LIN {X 0,Y 304.577,Z 613.756,A -85,B 0,C 180,E1 -15941.986,E2 -15941.986} C_VEL
LIN {X 0,Y 305.536,Z 607.014,A -85,B 0,C 180,E1 -15944.657,E2 -15944.657} C_VEL
LIN {X 0,Y 306.864,Z 599.737,A -85,B 0,C 180,E1 -15946.978,E2 -15946.978} C_VEL
LIN {X 0,Y 308.524,Z 590.973,A -85,B 0,C 180,E1 -15949.287,E2 -15949.287} C_VEL
LIN {X 0,Y 310.431,Z 582.076,A -85,B 0,C 180,E1 -15951.237,E2 -15951.237} C_VEL
LIN {X 0,Y 312.411,Z 571.551,A -85,B 0,C 180,E1 -15953.184,E2 -15953.184} C_VEL
LIN {X 0,Y 314.648,Z 560.119,A -85,B 0,C 180,E1 -15954.935,E2 -15954.935} C_VEL
LIN {X 0,Y 316.992,Z 547.692,A -85,B 0,C 180,E1 -15956.499,E2 -15956.499} C_VEL
LIN {X 0,Y 319.156,Z 534.543,A -85,B 0,C 180,E1 -15957.854,E2 -15957.854} C_VEL
LIN {X 0,Y 321.209,Z 520.123,A -85,B 0,C 180,E1 -15959.042,E2 -15959.042} C_VEL
LIN {X 0,Y 322.937,Z 505.843,A -85,B 0,C 180,E1 -15959.946,E2 -15959.946} C_VEL
LIN {X 0,Y 324.415,Z 490.603,A -85,B 0,C 180,E1 -15960.648,E2 -15960.648} C_VEL
LIN {X 0,Y 325.39,Z 474.711,A -85,B 0,C 180,E1 -15961.132,E2 -15961.132} C_VEL
LIN {X 0,Y 329.171,Z 367.113,A -85,B 0,C 180,E1 -15963.574,E2 -15963.574} C_VEL
LIN {X 0,Y 326.556,Z 352.02,A -85,B 0,C 180,E1 -15964.25,E2 -15964.25} C_VEL
LIN {X 0,Y 317.025,Z 330.376,A -85,B 0,C 180,E1 -15965.899,E2 -15965.899} C_VEL
LIN {X 0,Y 309.608,Z 314.884,A -85,B 0,C 180,E1 -15967.238,E2 -15967.238} C_VEL
LIN {X 0,Y 306.205,Z 302.97,A -85,B 0,C 180,E1 -15970.761,E2 -15970.761} C_VEL
LIN {X 0,Y 305.417,Z 300.068,A -85,B 0,C 180,E1 -15971.691,E2 -15971.691} C_VEL
LIN {X 0,Y 305.401,Z 300.067,A -85,B 0,C 180,E1 -15975.51,E2 -15975.51} C_VEL
LIN {X 0,Y 305.413,Z 300.072,A -85,B 0,C 180,E1 -15978.137,E2 -15978.137} C_VEL
LIN {X 0,Y 305.443,Z 300.059,A -85,B 0,C 180,E1 -15981.591,E2 -15981.591} C_VEL
LIN {X 0,Y 305.462,Z 300.049,A -85,B 0,C 180,E1 -15984.885,E2 -15984.885} C_VEL
LIN {X 0,Y 305.443,Z 300.063,A -85,B 0,C 180,E1 -15988.357,E2 -15988.357} C_VEL
LIN {X 0,Y 305.461,Z 300.061,A -85,B 0,C 180,E1 -15991.106,E2 -15991.106} C_VEL
LIN {X 0,Y 305.479,Z 300.062,A -85,B 0,C 180,E1 -15994.078,E2 -15994.078} C_VEL
LIN {X 0,Y 305.462,Z 300.065,A -85,B 0,C 180,E1 -15998.398,E2 -15998.398} C_VEL
LIN {X 0,Y 305.534,Z 300.055,A -85,B 0,C 180,E1 -16002.599,E2 -16002.599} C_VEL
LIN {X 0,Y 305.624,Z 300.022,A -85,B 0,C 180,E1 -16005.346,E2 -16005.346} C_VEL
LIN {X 0,Y 305.619,Z 300.022,A -85,B 0,C 180,E1 -16009.397,E2 -16009.397} C_VEL
LIN {X 0,Y 305.735,Z 300.026,A -85,B 0,C 180,E1 -16012.07,E2 -16012.07} C_VEL
LIN {X 0,Y 305.648,Z 300.023,A -85,B 0,C 180,E1 -16014.721,E2 -16014.721} C_VEL
LIN {X 0,Y 305.935,Z 299.985,A -85,B 0,C 180,E1 -16018.682,E2 -16018.682} C_VEL
LIN {X 0,Y 305.929,Z 300.002,A -85,B 0,C 180,E1 -16021.314,E2 -16021.314} C_VEL
LIN {X 0,Y 305.642,Z 300.007,A -85,B 0,C 180,E1 -16025.275,E2 -16025.275} C_VEL
LIN {X 0,Y 305.726,Z 299.997,A -85,B 0,C 180,E1 -16027.926,E2 -16027.926} C_VEL
LIN {X 0,Y 305.588,Z 300.044,A -85,B 0,C 180,E1 -16031.943,E2 -16031.943} C_VEL
LIN {X 0,Y 305.601,Z 300.02,A -85,B 0,C 180,E1 -16035.011,E2 -16035.011} C_VEL
LIN {X 0,Y 305.534,Z 300.035,A -85,B 0,C 180,E1 -16039.424,E2 -16039.424} C_VEL
LIN {X 0,Y 305.447,Z 300.062,A -85,B 0,C 180,E1 -16043.023,E2 -16043.023} C_VEL
LIN {X 0,Y 305.44,Z 300.031,A -85,B 0,C 180,E1 -16046.187,E2 -16046.187} C_VEL
LIN {X 0,Y 305.413,Z 300.045,A -85,B 0,C 180,E1 -16049.023,E2 -16049.023} C_VEL
LIN {X 0,Y 305.425,Z 300.064,A -85,B 0,C 180,E1 -16051.951,E2 -16051.951} C_VEL
LIN {X 0,Y 305.449,Z 300.04,A -85,B 0,C 180,E1 -16055.112,E2 -16055.112} C_VEL
LIN {X 0,Y 305.421,Z 300.049,A -85,B 0,C 180,E1 -16058.523,E2 -16058.523} C_VEL
LIN {X 0,Y 305.422,Z 300.064,A -85,B 0,C 180,E1 -16062.58,E2 -16062.58} C_VEL
LIN {X 0,Y 305.411,Z 300.047,A -85,B 0,C 180,E1 -16066.343,E2 -16066.343} C_VEL
LIN {X 0,Y 305.444,Z 300.063,A -85,B 0,C 180,E1 -16069.891,E2 -16069.891} C_VEL
LIN {X 0,Y 305.45,Z 300.044,A -85,B 0,C 180,E1 -16073.634,E2 -16073.634} C_VEL
LIN {X 0,Y 305.45,Z 300.064,A -85,B 0,C 180,E1 -16076.482,E2 -16076.482} C_VEL
LIN {X 0,Y 305.465,Z 300.05,A -85,B 0,C 180,E1 -16080.954,E2 -16080.954} C_VEL
LIN {X 0,Y 305.555,Z 300.041,A -85,B 0,C 180,E1 -16084.087,E2 -16084.087} C_VEL
LIN {X 0,Y 305.466,Z 300.058,A -85,B 0,C 180,E1 -16088.4,E2 -16088.4} C_VEL
LIN {X 0,Y 305.564,Z 300.051,A -85,B 0,C 180,E1 -16091.216,E2 -16091.216} C_VEL
LIN {X 0,Y 305.633,Z 300.039,A -85,B 0,C 180,E1 -16095.348,E2 -16095.348} C_VEL
LIN {X 0,Y 305.624,Z 300.035,A -85,B 0,C 180,E1 -16099.399,E2 -16099.399} C_VEL
LIN {X 0,Y 305.807,Z 300.029,A -85,B 0,C 180,E1 -16102.323,E2 -16102.323} C_VEL
LIN {X 0,Y 306.955,Z 303.051,A -85,B 0,C 180,E1 -16102.591,E2 -16102.591} C_VEL
LIN {X 0,Y 308.436,Z 305.417,A -85,B 0,C 180,E1 -16102.849,E2 -16102.849} C_VEL
LIN {X 0,Y 312.255,Z 312.818,A -85,B 0,C 180,E1 -16103.538,E2 -16103.538} C_VEL
LIN {X 0,Y 320.275,Z 328.458,A -85,B 0,C 180,E1 -16104.919,E2 -16104.919} C_VEL
LIN {X 0,Y 327.005,Z 343.478,A -85,B 0,C 180,E1 -16106.065,E2 -16106.065} C_VEL
LIN {X 0,Y 329.522,Z 349.607,A -85,B 0,C 180,E1 -16106.495,E2 -16106.495} C_VEL
LIN {X 0,Y 325.777,Z 455.006,A -85,B 0,C 180,E1 -16108.879,E2 -16108.879} C_VEL
LIN {X 0,Y 324.99,Z 471.109,A -85,B 0,C 180,E1 -16109.341,E2 -16109.341} C_VEL
LIN {X 0,Y 323.73,Z 486.619,A -85,B 0,C 180,E1 -16110.029,E2 -16110.029} C_VEL
LIN {X 0,Y 322.104,Z 501.197,A -85,B 0,C 180,E1 -16110.922,E2 -16110.922} C_VEL
LIN {X 0,Y 320.359,Z 515.115,A -85,B 0,C 180,E1 -16112.042,E2 -16112.042} C_VEL
LIN {X 0,Y 318.327,Z 527.994,A -85,B 0,C 180,E1 -16113.322,E2 -16113.322} C_VEL
LIN {X 0,Y 316.161,Z 540.387,A -85,B 0,C 180,E1 -16114.828,E2 -16114.828} C_VEL
LIN {X 0,Y 313.949,Z 552.293,A -85,B 0,C 180,E1 -16116.587,E2 -16116.587} C_VEL
LIN {X 0,Y 311.841,Z 562.917,A -85,B 0,C 180,E1 -16118.476,E2 -16118.476} C_VEL
LIN {X 0,Y 309.656,Z 573.654,A -85,B 0,C 180,E1 -16120.791,E2 -16120.791} C_VEL
LIN {X 0,Y 307.746,Z 582.782,A -85,B 0,C 180,E1 -16123.2,E2 -16123.2} C_VEL
LIN {X 0,Y 306.329,Z 589.979,A -85,B 0,C 180,E1 -16125.521,E2 -16125.521} C_VEL
LIN {X 0,Y 305.184,Z 596.469,A -85,B 0,C 180,E1 -16128.112,E2 -16128.112} C_VEL
LIN {X 0,Y 304.506,Z 600.773,A -85,B 0,C 180,E1 -16130.254,E2 -16130.254} C_VEL
LIN {X 0,Y 304.024,Z 604.144,A -85,B 0,C 180,E1 -16132.391,E2 -16132.391} C_VEL
LIN {X 0,Y 303.484,Z 607.573,A -85,B 0,C 180,E1 -16135.432,E2 -16135.432} C_VEL
LIN {X 0,Y 303.276,Z 609.377,A -85,B 0,C 180,E1 -16138.292,E2 -16138.292} C_VEL
LIN {X 0,Y 303.287,Z 609.865,A -85,B 0,C 180,E1 -16140.981,E2 -16140.981} C_VEL
LIN {X 0,Y 303.443,Z 609.138,A -85,B 0,C 180,E1 -16143.768,E2 -16143.768} C_VEL
LIN {X 0,Y 303.721,Z 607.678,A -85,B 0,C 180,E1 -16145.92,E2 -16145.92} C_VEL
LIN {X 0,Y 304.272,Z 604.832,A -85,B 0,C 180,E1 -16148.581,E2 -16148.581} C_VEL
LIN {X 0,Y 305.088,Z 600.978,A -85,B 0,C 180,E1 -16151.117,E2 -16151.117} C_VEL
LIN {X 0,Y 306.161,Z 596.204,A -85,B 0,C 180,E1 -16153.522,E2 -16153.522} C_VEL
LIN {X 0,Y 307.867,Z 588.815,A -85,B 0,C 180,E1 -16156.419,E2 -16156.419} C_VEL
LIN {X 0,Y 309.828,Z 580.921,A -85,B 0,C 180,E1 -16158.87,E2 -16158.87} C_VEL
LIN {X 0,Y 312.17,Z 571.322,A -85,B 0,C 180,E1 -16161.289,E2 -16161.289} C_VEL
LIN {X 0,Y 314.85,Z 560.656,A -85,B 0,C 180,E1 -16163.471,E2 -16163.471} C_VEL
LIN {X 0,Y 315.34,Z 558.594,A -85,B 0,C 180,E1 -16163.84,E2 -16163.84} C_VEL
LIN {X 0,Y 315.768,Z 554.512,A -85,B 0,C 180,E1 -16164.61,E2 -16164.61} C_VEL
LIN {X 0,Y 314.792,Z 547.859,A -85,B 0,C 180,E1 -16165.94,E2 -16165.94} C_VEL
LIN {X 0,Y 313.825,Z 540.87,A -85,B 0,C 180,E1 -16167.207,E2 -16167.207} C_VEL
LIN {X 0,Y 314.234,Z 536.226,A -85,B 0,C 180,E1 -16167.866,E2 -16167.866} C_VEL
LIN {X 0,Y 316.764,Z 523.451,A -85,B 0,C 180,E1 -16169.319,E2 -16169.319} C_VEL
LIN {X 0,Y 319.172,Z 509.538,A -85,B 0,C 180,E1 -16170.589,E2 -16170.589} C_VEL
LIN {X 0,Y 321.16,Z 495.876,A -85,B 0,C 180,E1 -16171.57,E2 -16171.57} C_VEL
LIN {X 0,Y 322.848,Z 481.049,A -85,B 0,C 180,E1 -16172.378,E2 -16172.378} C_VEL
LIN {X 0,Y 324.161,Z 465.241,A -85,B 0,C 180,E1 -16172.968,E2 -16172.968} C_VEL
LIN {X 0,Y 329.009,Z 355.514,A -85,B 0,C 180,E1 -16175.564,E2 -16175.564} C_VEL
LIN {X 0,Y 322.304,Z 340.991,A -85,B 0,C 180,E1 -16177.02,E2 -16177.02} C_VEL
LIN {X 0,Y 315.332,Z 328.219,A -85,B 0,C 180,E1 -16178.583,E2 -16178.583} C_VEL
LIN {X 0,Y 308.492,Z 316.768,A -85,B 0,C 180,E1 -16180.219,E2 -16180.219} C_VEL
LIN {X 0,Y 301.733,Z 306.632,A -85,B 0,C 180,E1 -16181.938,E2 -16181.938} C_VEL
LIN {X 0,Y 299.049,Z 302.887,A -85,B 0,C 180,E1 -16182.655,E2 -16182.655} C_VEL
LIN {X 0,Y 298.75,Z 302.016,A -85,B 0,C 180,E1 -16182.902,E2 -16182.902} C_VEL
LIN {X 0,Y 298.506,Z 300.928,A -85,B 0,C 180,E1 -16183.416,E2 -16183.416} C_VEL
LIN {X 0,Y 298.54,Z 300.924,A -85,B 0,C 180,E1 -16186.387,E2 -16186.387} C_VEL
LIN {X 0,Y 298.717,Z 300.898,A -85,B 0,C 180,E1 -16191.157,E2 -16191.157} C_VEL
LIN {X 0,Y 298.776,Z 300.891,A -85,B 0,C 180,E1 -16193.248,E2 -16193.248} C_VEL
LIN {X 0,Y 298.913,Z 300.873,A -85,B 0,C 180,E1 -16198.655,E2 -16198.655} C_VEL
LIN {X 0,Y 298.913,Z 300.872,A -85,B 0,C 180,E1 -16201.349,E2 -16201.349} C_VEL
LIN {X 0,Y 298.632,Z 300.907,A -85,B 0,C 180,E1 -16205.404,E2 -16205.404} C_VEL
LIN {X 0,Y 298.701,Z 300.895,A -85,B 0,C 180,E1 -16208.118,E2 -16208.118} C_VEL
LIN {X 0,Y 298.542,Z 300.922,A -85,B 0,C 180,E1 -16212.234,E2 -16212.234} C_VEL
LIN {X 0,Y 298.542,Z 300.922,A -85,B 0,C 180,E1 -16215.17,E2 -16215.17} C_VEL
LIN {X 0,Y 298.436,Z 300.931,A -85,B 0,C 180,E1 -16219.619,E2 -16219.619} C_VEL
LIN {X 0,Y 298.383,Z 300.937,A -85,B 0,C 180,E1 -16223.606,E2 -16223.606} C_VEL
LIN {X 0,Y 298.397,Z 300.935,A -85,B 0,C 180,E1 -16226.585,E2 -16226.585} C_VEL
LIN {X 0,Y 298.352,Z 300.941,A -85,B 0,C 180,E1 -16229.65,E2 -16229.65} C_VEL
LIN {X 0,Y 298.388,Z 300.941,A -85,B 0,C 180,E1 -16232.803,E2 -16232.803} C_VEL
LIN {X 0,Y 298.4,Z 300.936,A -85,B 0,C 180,E1 -16236.074,E2 -16236.074} C_VEL
LIN {X 0,Y 298.372,Z 300.938,A -85,B 0,C 180,E1 -16239.494,E2 -16239.494} C_VEL
LIN {X 0,Y 298.367,Z 300.944,A -85,B 0,C 180,E1 -16243.191,E2 -16243.191} C_VEL
LIN {X 0,Y 301.448,Z 310.139,A -85,B 0,C 180,E1 -16247.022,E2 -16247.022} C_VEL
LIN {X 0,Y 302.439,Z 313.009,A -85,B 0,C 180,E1 -16248.08,E2 -16248.08} C_VEL
LIN {X 0,Y 305.018,Z 317.369,A -85,B 0,C 180,E1 -16248.765,E2 -16248.765} C_VEL
LIN {X 0,Y 309.62,Z 324.965,A -85,B 0,C 180,E1 -16249.913,E2 -16249.913} C_VEL
LIN {X 0,Y 316.602,Z 337.504,A -85,B 0,C 180,E1 -16251.572,E2 -16251.572} C_VEL
LIN {X 0,Y 323.262,Z 351.325,A -85,B 0,C 180,E1 -16253.086,E2 -16253.086} C_VEL
LIN {X 0,Y 327.305,Z 360.726,A -85,B 0,C 180,E1 -16253.978,E2 -16253.978} C_VEL
LIN {X 0,Y 328.618,Z 369.992,A -85,B 0,C 180,E1 -16254.444,E2 -16254.444} C_VEL
LIN {X 0,Y 323.645,Z 480.078,A -85,B 0,C 180,E1 -16257.029,E2 -16257.029} C_VEL
LIN {X 0,Y 322.213,Z 495.821,A -85,B 0,C 180,E1 -16257.607,E2 -16257.607} C_VEL
LIN {X 0,Y 320.261,Z 510.942,A -85,B 0,C 180,E1 -16258.405,E2 -16258.405} C_VEL
LIN {X 0,Y 318.016,Z 525.542,A -85,B 0,C 180,E1 -16259.451,E2 -16259.451} C_VEL
LIN {X 0,Y 315.545,Z 538.838,A -85,B 0,C 180,E1 -16260.661,E2 -16260.661} C_VEL
LIN {X 0,Y 312.73,Z 552.45,A -85,B 0,C 180,E1 -16262.206,E2 -16262.206} C_VEL
LIN {X 0,Y 309.812,Z 564.833,A -85,B 0,C 180,E1 -16263.928,E2 -16263.928} C_VEL
LIN {X 0,Y 307.265,Z 575.247,A -85,B 0,C 180,E1 -16265.689,E2 -16265.689} C_VEL
LIN {X 0,Y 304.896,Z 584.966,A -85,B 0,C 180,E1 -16267.652,E2 -16267.652} C_VEL
LIN {X 0,Y 302.404,Z 594.512,A -85,B 0,C 180,E1 -16269.954,E2 -16269.954} C_VEL
LIN {X 0,Y 300.222,Z 603.53,A -85,B 0,C 180,E1 -16272.635,E2 -16272.635} C_VEL
LIN {X 0,Y 298.778,Z 609.997,A -85,B 0,C 180,E1 -16275.005,E2 -16275.005} C_VEL
LIN {X 0,Y 297.647,Z 615.964,A -85,B 0,C 180,E1 -16277.732,E2 -16277.732} C_VEL
LIN {X 0,Y 296.915,Z 620.57,A -85,B 0,C 180,E1 -16280.463,E2 -16280.463} C_VEL
LIN {X 0,Y 296.549,Z 623.898,A -85,B 0,C 180,E1 -16283.195,E2 -16283.195} C_VEL
LIN {X 0,Y 296.458,Z 625.984,A -85,B 0,C 180,E1 -16285.922,E2 -16285.922} C_VEL
LIN {X 0,Y 296.492,Z 626.905,A -85,B 0,C 180,E1 -16288.642,E2 -16288.642} C_VEL
LIN {X 0,Y 296.493,Z 626.666,A -85,B 0,C 180,E1 -16291.359,E2 -16291.359} C_VEL
LIN {X 0,Y 296.474,Z 625.255,A -85,B 0,C 180,E1 -16294.079,E2 -16294.079} C_VEL
LIN {X 0,Y 296.558,Z 622.628,A -85,B 0,C 180,E1 -16296.806,E2 -16296.806} C_VEL
LIN {X 0,Y 296.898,Z 618.702,A -85,B 0,C 180,E1 -16299.538,E2 -16299.538} C_VEL
LIN {X 0,Y 297.558,Z 613.417,A -85,B 0,C 180,E1 -16302.273,E2 -16302.273} C_VEL
LIN {X 0,Y 298.592,Z 606.638,A -85,B 0,C 180,E1 -16305.006,E2 -16305.006} C_VEL
LIN {X 0,Y 300.003,Z 599.318,A -85,B 0,C 180,E1 -16307.379,E2 -16307.379} C_VEL
LIN {X 0,Y 301.747,Z 590.506,A -85,B 0,C 180,E1 -16309.738,E2 -16309.738} C_VEL
LIN {X 0,Y 303.682,Z 581.548,A -85,B 0,C 180,E1 -16311.733,E2 -16311.733} C_VEL
LIN {X 0,Y 305.786,Z 570.96,A -85,B 0,C 180,E1 -16313.716,E2 -16313.716} C_VEL
LIN {X 0,Y 308.177,Z 559.453,A -85,B 0,C 180,E1 -16315.496,E2 -16315.496} C_VEL
LIN {X 0,Y 310.567,Z 546.933,A -85,B 0,C 180,E1 -16317.092,E2 -16317.092} C_VEL
LIN {X 0,Y 312.98,Z 532.703,A -85,B 0,C 180,E1 -16318.555,E2 -16318.555} C_VEL
LIN {X 0,Y 315.088,Z 517.922,A -85,B 0,C 180,E1 -16319.754,E2 -16319.754} C_VEL
LIN {X 0,Y 316.909,Z 503.043,A -85,B 0,C 180,E1 -16320.668,E2 -16320.668} C_VEL
LIN {X 0,Y 318.362,Z 487.666,A -85,B 0,C 180,E1 -16321.342,E2 -16321.342} C_VEL
LIN {X 0,Y 319.261,Z 471.708,A -85,B 0,C 180,E1 -16321.799,E2 -16321.799} C_VEL
LIN {X 0,Y 323.041,Z 368.125,A -85,B 0,C 180,E1 -16324.19,E2 -16324.19} C_VEL
LIN {X 0,Y 320.673,Z 354.538,A -85,B 0,C 180,E1 -16324.816,E2 -16324.816} C_VEL
LIN {X 0,Y 311.45,Z 333.628,A -85,B 0,C 180,E1 -16326.462,E2 -16326.462} C_VEL
LIN {X 0,Y 303.958,Z 318.2,A -85,B 0,C 180,E1 -16327.841,E2 -16327.841} C_VEL
LIN {X 0,Y 302.264,Z 314.622,A -85,B 0,C 180,E1 -16328.184,E2 -16328.184} C_VEL
LIN {X 0,Y 298.993,Z 303.051,A -85,B 0,C 180,E1 -16331.727,E2 -16331.727} C_VEL
LIN {X 0,Y 298.401,Z 300.936,A -85,B 0,C 180,E1 -16332.463,E2 -16332.463} C_VEL
LIN {X 0,Y 298.371,Z 300.937,A -85,B 0,C 180,E1 -16336.913,E2 -16336.913} C_VEL
LIN {X 0,Y 298.387,Z 300.934,A -85,B 0,C 180,E1 -16341.01,E2 -16341.01} C_VEL
LIN {X 0,Y 298.405,Z 300.938,A -85,B 0,C 180,E1 -16343.926,E2 -16343.926} C_VEL
LIN {X 0,Y 298.394,Z 300.937,A -85,B 0,C 180,E1 -16347.198,E2 -16347.198} C_VEL
LIN {X 0,Y 298.369,Z 300.944,A -85,B 0,C 180,E1 -16350.635,E2 -16350.635} C_VEL
LIN {X 0,Y 298.413,Z 300.941,A -85,B 0,C 180,E1 -16354.916,E2 -16354.916} C_VEL
LIN {X 0,Y 298.394,Z 300.946,A -85,B 0,C 180,E1 -16357.86,E2 -16357.86} C_VEL
LIN {X 0,Y 298.463,Z 300.929,A -85,B 0,C 180,E1 -16360.75,E2 -16360.75} C_VEL
LIN {X 0,Y 298.585,Z 300.904,A -85,B 0,C 180,E1 -16364.992,E2 -16364.992} C_VEL
LIN {X 0,Y 298.578,Z 300.897,A -85,B 0,C 180,E1 -16369.144,E2 -16369.144} C_VEL
LIN {X 0,Y 298.681,Z 300.906,A -85,B 0,C 180,E1 -16371.882,E2 -16371.882} C_VEL
LIN {X 0,Y 298.618,Z 300.9,A -85,B 0,C 180,E1 -16374.596,E2 -16374.596} C_VEL
LIN {X 0,Y 298.902,Z 300.86,A -85,B 0,C 180,E1 -16378.651,E2 -16378.651} C_VEL
LIN {X 0,Y 298.897,Z 300.878,A -85,B 0,C 180,E1 -16381.345,E2 -16381.345} C_VEL
LIN {X 0,Y 298.68,Z 300.864,A -85,B 0,C 180,E1 -16386.51,E2 -16386.51} C_VEL
LIN {X 0,Y 298.609,Z 300.901,A -85,B 0,C 180,E1 -16389.48,E2 -16389.48} C_VEL
LIN {X 0,Y 298.536,Z 300.914,A -85,B 0,C 180,E1 -16393.614,E2 -16393.614} C_VEL
LIN {X 0,Y 298.477,Z 300.892,A -85,B 0,C 180,E1 -16396.41,E2 -16396.41} C_VEL
LIN {X 0,Y 298.47,Z 300.917,A -85,B 0,C 180,E1 -16399.634,E2 -16399.634} C_VEL
LIN {X 0,Y 298.378,Z 300.936,A -85,B 0,C 180,E1 -16403.601,E2 -16403.601} C_VEL
LIN {X 0,Y 298.391,Z 300.905,A -85,B 0,C 180,E1 -16406.581,E2 -16406.581} C_VEL
LIN {X 0,Y 298.346,Z 300.933,A -85,B 0,C 180,E1 -16409.646,E2 -16409.646} C_VEL
LIN {X 0,Y 298.382,Z 300.943,A -85,B 0,C 180,E1 -16412.799,E2 -16412.799} C_VEL
LIN {X 0,Y 298.391,Z 300.91,A -85,B 0,C 180,E1 -16416.07,E2 -16416.07} C_VEL
LIN {X 0,Y 298.361,Z 300.938,A -85,B 0,C 180,E1 -16419.49,E2 -16419.49} C_VEL
LIN {X 0,Y 298.357,Z 300.937,A -85,B 0,C 180,E1 -16423.095,E2 -16423.095} C_VEL
LIN {X 0,Y 298.39,Z 300.926,A -85,B 0,C 180,E1 -16426.919,E2 -16426.919} C_VEL
LIN {X 0,Y 298.385,Z 300.936,A -85,B 0,C 180,E1 -16431.006,E2 -16431.006} C_VEL
LIN {X 0,Y 298.392,Z 300.925,A -85,B 0,C 180,E1 -16433.927,E2 -16433.927} C_VEL
LIN {X 0,Y 298.378,Z 300.942,A -85,B 0,C 180,E1 -16437.198,E2 -16437.198} C_VEL
LIN {X 0,Y 298.441,Z 300.934,A -85,B 0,C 180,E1 -16441.902,E2 -16441.902} C_VEL
LIN {X 0,Y 298.468,Z 300.919,A -85,B 0,C 180,E1 -16444.922,E2 -16444.922} C_VEL
LIN {X 0,Y 298.421,Z 300.928,A -85,B 0,C 180,E1 -16449.313,E2 -16449.313} C_VEL
LIN {X 0,Y 298.518,Z 300.927,A -85,B 0,C 180,E1 -16452.178,E2 -16452.178} C_VEL
LIN {X 0,Y 298.578,Z 300.92,A -85,B 0,C 180,E1 -16454.994,E2 -16454.994} C_VEL
LIN {X 0,Y 298.579,Z 300.913,A -85,B 0,C 180,E1 -16459.146,E2 -16459.146} C_VEL
LIN {X 0,Y 298.752,Z 301.04,A -85,B 0,C 180,E1 -16461.458,E2 -16461.458} C_VEL
LIN {X 0,Y 299.802,Z 303.851,A -85,B 0,C 180,E1 -16461.685,E2 -16461.685} C_VEL
LIN {X 0,Y 301.221,Z 305.91,A -85,B 0,C 180,E1 -16461.935,E2 -16461.935} C_VEL
LIN {X 0,Y 306.216,Z 314.852,A -85,B 0,C 180,E1 -16462.846,E2 -16462.846} C_VEL
LIN {X 0,Y 315.744,Z 333.935,A -85,B 0,C 180,E1 -16464.554,E2 -16464.554} C_VEL
LIN {X 0,Y 321.991,Z 348.108,A -85,B 0,C 180,E1 -16465.651,E2 -16465.651} C_VEL
LIN {X 0,Y 323.327,Z 351.429,A -85,B 0,C 180,E1 -16465.887,E2 -16465.887} C_VEL
LIN {X 0,Y 320.967,Z 417.187,A -85,B 0,C 180,E1 -16467.409,E2 -16467.409} C_VEL
LIN {X 0,Y 319.116,Z 465.131,A -85,B 0,C 180,E1 -16468.54,E2 -16468.54} C_VEL
LIN {X 0,Y 317.931,Z 481.286,A -85,B 0,C 180,E1 -16469.168,E2 -16469.168} C_VEL
LIN {X 0,Y 316.46,Z 496.082,A -85,B 0,C 180,E1 -16469.999,E2 -16469.999} C_VEL
LIN {X 0,Y 314.722,Z 509.849,A -85,B 0,C 180,E1 -16471.015,E2 -16471.015} C_VEL
LIN {X 0,Y 312.445,Z 524.72,A -85,B 0,C 180,E1 -16472.417,E2 -16472.417} C_VEL
LIN {X 0,Y 310.257,Z 537.349,A -85,B 0,C 180,E1 -16473.896,E2 -16473.896} C_VEL
LIN {X 0,Y 308.023,Z 549.06,A -85,B 0,C 180,E1 -16475.564,E2 -16475.564} C_VEL
LIN {X 0,Y 305.597,Z 560.862,A -85,B 0,C 180,E1 -16477.598,E2 -16477.598} C_VEL
LIN {X 0,Y 303.513,Z 570.735,A -85,B 0,C 180,E1 -16479.664,E2 -16479.664} C_VEL
LIN {X 0,Y 301.401,Z 580.417,A -85,B 0,C 180,E1 -16482.113,E2 -16482.113} C_VEL
LIN {X 0,Y 299.762,Z 588.387,A -85,B 0,C 180,E1 -16484.597,E2 -16484.597} C_VEL
LIN {X 0,Y 298.502,Z 594.928,A -85,B 0,C 180,E1 -16487.115,E2 -16487.115} C_VEL
LIN {X 0,Y 297.469,Z 600.883,A -85,B 0,C 180,E1 -16490.033,E2 -16490.033} C_VEL
LIN {X 0,Y 296.891,Z 604.797,A -85,B 0,C 180,E1 -16492.609,E2 -16492.609} C_VEL
LIN {X 0,Y 296.374,Z 608.046,A -85,B 0,C 180,E1 -16495.704,E2 -16495.704} C_VEL
LIN {X 0,Y 296.179,Z 609.692,A -85,B 0,C 180,E1 -16498.609,E2 -16498.609} C_VEL
LIN {X 0,Y 296.202,Z 610.031,A -85,B 0,C 180,E1 -16501.465,E2 -16501.465} C_VEL
LIN {X 0,Y 296.358,Z 609.352,A -85,B 0,C 180,E1 -16503.906,E2 -16503.906} C_VEL
LIN {X 0,Y 296.695,Z 607.697,A -85,B 0,C 180,E1 -16506.358,E2 -16506.358} C_VEL
LIN {X 0,Y 297.222,Z 605.213,A -85,B 0,C 180,E1 -16508.716,E2 -16508.716} C_VEL
LIN {X 0,Y 298.074,Z 601.433,A -85,B 0,C 180,E1 -16511.312,E2 -16511.312} C_VEL
LIN {X 0,Y 299.268,Z 596.423,A -85,B 0,C 180,E1 -16513.903,E2 -16513.903} C_VEL
LIN {X 0,Y 300.767,Z 590.26,A -85,B 0,C 180,E1 -16516.415,E2 -16516.415} C_VEL
LIN {X 0,Y 302.667,Z 582.896,A -85,B 0,C 180,E1 -16518.843,E2 -16518.843} C_VEL
LIN {X 0,Y 304.827,Z 574.624,A -85,B 0,C 180,E1 -16521.087,E2 -16521.087} C_VEL
LIN {X 0,Y 307.279,Z 565.354,A -85,B 0,C 180,E1 -16523.176,E2 -16523.176} C_VEL
LIN {X 0,Y 309.977,Z 554.576,A -85,B 0,C 180,E1 -16525.191,E2 -16525.191} C_VEL
LIN {X 0,Y 312.761,Z 542.792,A -85,B 0,C 180,E1 -16527.002,E2 -16527.002} C_VEL
LIN {X 0,Y 314.234,Z 536.226,A -85,B 0,C 180,E1 -16527.866,E2 -16527.866} C_VEL
LIN {X 0,Y 314.679,Z 531.511,A -85,B 0,C 180,E1 -16528.505,E2 -16528.505} C_VEL
LIN {X 0,Y 312.936,Z 517.527,A -85,B 0,C 180,E1 -16530.511,E2 -16530.511} C_VEL
LIN {X 0,Y 312.932,Z 512.493,A -85,B 0,C 180,E1 -16531.075,E2 -16531.075} C_VEL
LIN {X 0,Y 313.144,Z 510.739,A -85,B 0,C 180,E1 -16531.234,E2 -16531.234} C_VEL
LIN {X 0,Y 315.284,Z 496.831,A -85,B 0,C 180,E1 -16532.265,E2 -16532.265} C_VEL
LIN {X 0,Y 317.091,Z 481.788,A -85,B 0,C 180,E1 -16533.106,E2 -16533.106} C_VEL
LIN {X 0,Y 318.456,Z 466.059,A -85,B 0,C 180,E1 -16533.712,E2 -16533.712} C_VEL
LIN {X 0,Y 323.51,Z 357.908,A -85,B 0,C 180,E1 -16536.303,E2 -16536.303} C_VEL
LIN {X 0,Y 317.125,Z 344.104,A -85,B 0,C 180,E1 -16537.757,E2 -16537.757} C_VEL
LIN {X 0,Y 310.479,Z 331.816,A -85,B 0,C 180,E1 -16539.322,E2 -16539.322} C_VEL
LIN {X 0,Y 304.375,Z 321.582,A -85,B 0,C 180,E1 -16540.839,E2 -16540.839} C_VEL
LIN {X 0,Y 298.095,Z 311.954,A -85,B 0,C 180,E1 -16542.509,E2 -16542.509} C_VEL
LIN {X 0,Y 295.349,Z 308.029,A -85,B 0,C 180,E1 -16543.278,E2 -16543.278} C_VEL
LIN {X 0,Y 292.175,Z 304.061,A -85,B 0,C 180,E1 -16544.182,E2 -16544.182} C_VEL
LIN {X 0,Y 291.703,Z 302.754,A -85,B 0,C 180,E1 -16544.366,E2 -16544.366} C_VEL
LIN {X 0,Y 291.53,Z 301.796,A -85,B 0,C 180,E1 -16544.853,E2 -16544.853} C_VEL
LIN {X 0,Y 291.524,Z 301.794,A -85,B 0,C 180,E1 -16548.883,E2 -16548.883} C_VEL
LIN {X 0,Y 291.677,Z 301.774,A -85,B 0,C 180,E1 -16551.69,E2 -16551.69} C_VEL
LIN {X 0,Y 291.616,Z 301.782,A -85,B 0,C 180,E1 -16554.47,E2 -16554.47} C_VEL
LIN {X 0,Y 291.879,Z 301.749,A -85,B 0,C 180,E1 -16558.623,E2 -16558.623} C_VEL
LIN {X 0,Y 291.879,Z 301.748,A -85,B 0,C 180,E1 -16561.382,E2 -16561.382} C_VEL
LIN {X 0,Y 291.69,Z 301.774,A -85,B 0,C 180,E1 -16566.921,E2 -16566.921} C_VEL
LIN {X 0,Y 291.561,Z 301.792,A -85,B 0,C 180,E1 -16569.716,E2 -16569.716} C_VEL
LIN {X 0,Y 291.508,Z 301.792,A -85,B 0,C 180,E1 -16573.953,E2 -16573.953} C_VEL
LIN {X 0,Y 291.422,Z 301.803,A -85,B 0,C 180,E1 -16576.824,E2 -16576.824} C_VEL
LIN {X 0,Y 291.386,Z 301.808,A -85,B 0,C 180,E1 -16579.844,E2 -16579.844} C_VEL
LIN {X 0,Y 291.329,Z 301.819,A -85,B 0,C 180,E1 -16584.214,E2 -16584.214} C_VEL
LIN {X 0,Y 291.325,Z 301.821,A -85,B 0,C 180,E1 -16587.283,E2 -16587.283} C_VEL
LIN {X 0,Y 291.297,Z 301.823,A -85,B 0,C 180,E1 -16590.443,E2 -16590.443} C_VEL
LIN {X 0,Y 291.34,Z 301.814,A -85,B 0,C 180,E1 -16593.701,E2 -16593.701} C_VEL
LIN {X 0,Y 291.349,Z 301.813,A -85,B 0,C 180,E1 -16597.25,E2 -16597.25} C_VEL
LIN {X 0,Y 291.297,Z 301.824,A -85,B 0,C 180,E1 -16600.651,E2 -16600.651} C_VEL
LIN {X 0,Y 291.279,Z 301.841,A -85,B 0,C 180,E1 -16601.732,E2 -16601.732} C_VEL
LIN {X 0,Y 294.357,Z 310.811,A -85,B 0,C 180,E1 -16605.75,E2 -16605.75} C_VEL
LIN {X 0,Y 295.023,Z 312.656,A -85,B 0,C 180,E1 -16606.464,E2 -16606.464} C_VEL
LIN {X 0,Y 298.157,Z 317.586,A -85,B 0,C 180,E1 -16607.354,E2 -16607.354} C_VEL
LIN {X 0,Y 305.17,Z 329.137,A -85,B 0,C 180,E1 -16609.219,E2 -16609.219} C_VEL
LIN {X 0,Y 312.104,Z 341.803,A -85,B 0,C 180,E1 -16610.944,E2 -16610.944} C_VEL
LIN {X 0,Y 318.245,Z 354.662,A -85,B 0,C 180,E1 -16612.399,E2 -16612.399} C_VEL
LIN {X 0,Y 322.132,Z 363.873,A -85,B 0,C 180,E1 -16613.304,E2 -16613.304} C_VEL
LIN {X 0,Y 323.105,Z 370.767,A -85,B 0,C 180,E1 -16613.665,E2 -16613.665} C_VEL
LIN {X 0,Y 317.981,Z 479.986,A -85,B 0,C 180,E1 -16616.269,E2 -16616.269} C_VEL
LIN {X 0,Y 316.401,Z 496.403,A -85,B 0,C 180,E1 -16616.889,E2 -16616.889} C_VEL
LIN {X 0,Y 314.28,Z 511.836,A -85,B 0,C 180,E1 -16617.732,E2 -16617.732} C_VEL
LIN {X 0,Y 311.956,Z 526.16,A -85,B 0,C 180,E1 -16618.792,E2 -16618.792} C_VEL
LIN {X 0,Y 309.08,Z 540.738,A -85,B 0,C 180,E1 -16620.173,E2 -16620.173} C_VEL
LIN {X 0,Y 306.197,Z 553.958,A -85,B 0,C 180,E1 -16621.746,E2 -16621.746} C_VEL
LIN {X 0,Y 303.188,Z 566.071,A -85,B 0,C 180,E1 -16623.5,E2 -16623.5} C_VEL
LIN {X 0,Y 300.31,Z 577.338,A -85,B 0,C 180,E1 -16625.494,E2 -16625.494} C_VEL
LIN {X 0,Y 297.578,Z 587.982,A -85,B 0,C 180,E1 -16627.799,E2 -16627.799} C_VEL
LIN {X 0,Y 295.088,Z 597.016,A -85,B 0,C 180,E1 -16630.162,E2 -16630.162} C_VEL
LIN {X 0,Y 293.145,Z 604.536,A -85,B 0,C 180,E1 -16632.563,E2 -16632.563} C_VEL
LIN {X 0,Y 291.515,Z 611.584,A -85,B 0,C 180,E1 -16635.338,E2 -16635.338} C_VEL
LIN {X 0,Y 290.378,Z 617.146,A -85,B 0,C 180,E1 -16638.129,E2 -16638.129} C_VEL
LIN {X 0,Y 289.849,Z 620.45,A -85,B 0,C 180,E1 -16640.229,E2 -16640.229} C_VEL
LIN {X 0,Y 289.466,Z 623.759,A -85,B 0,C 180,E1 -16643.028,E2 -16643.028} C_VEL
LIN {X 0,Y 289.363,Z 625.816,A -85,B 0,C 180,E1 -16645.822,E2 -16645.822} C_VEL
LIN {X 0,Y 289.413,Z 626.708,A -85,B 0,C 180,E1 -16648.609,E2 -16648.609} C_VEL
LIN {X 0,Y 289.414,Z 626.441,A -85,B 0,C 180,E1 -16651.392,E2 -16651.392} C_VEL
LIN {X 0,Y 289.379,Z 625,A -85,B 0,C 180,E1 -16654.179,E2 -16654.179} C_VEL
LIN {X 0,Y 289.474,Z 622.351,A -85,B 0,C 180,E1 -16656.973,E2 -16656.973} C_VEL
LIN {X 0,Y 289.823,Z 618.397,A -85,B 0,C 180,E1 -16659.773,E2 -16659.773} C_VEL
LIN {X 0,Y 290.556,Z 613.075,A -85,B 0,C 180,E1 -16662.574,E2 -16662.574} C_VEL
LIN {X 0,Y 291.699,Z 605.979,A -85,B 0,C 180,E1 -16665.474,E2 -16665.474} C_VEL
LIN {X 0,Y 293.36,Z 597.741,A -85,B 0,C 180,E1 -16668.146,E2 -16668.146} C_VEL
LIN {X 0,Y 295.367,Z 588.636,A -85,B 0,C 180,E1 -16670.546,E2 -16670.546} C_VEL
LIN {X 0,Y 297.421,Z 578.785,A -85,B 0,C 180,E1 -16672.699,E2 -16672.699} C_VEL
LIN {X 0,Y 299.595,Z 568.324,A -85,B 0,C 180,E1 -16674.607,E2 -16674.607} C_VEL
LIN {X 0,Y 302.195,Z 556.329,A -85,B 0,C 180,E1 -16676.409,E2 -16676.409} C_VEL
LIN {X 0,Y 304.674,Z 543.179,A -85,B 0,C 180,E1 -16678.034,E2 -16678.034} C_VEL
LIN {X 0,Y 307.016,Z 529.495,A -85,B 0,C 180,E1 -16679.393,E2 -16679.393} C_VEL
LIN {X 0,Y 309.037,Z 515.545,A -85,B 0,C 180,E1 -16680.492,E2 -16680.492} C_VEL
LIN {X 0,Y 310.878,Z 500.69,A -85,B 0,C 180,E1 -16681.377,E2 -16681.377} C_VEL
LIN {X 0,Y 312.257,Z 485.397,A -85,B 0,C 180,E1 -16682.027,E2 -16682.027} C_VEL
LIN {X 0,Y 313.191,Z 466.628,A -85,B 0,C 180,E1 -16682.538,E2 -16682.538} C_VEL
LIN {X 0,Y 316.943,Z 369.141,A -85,B 0,C 180,E1 -16684.823,E2 -16684.823} C_VEL
LIN {X 0,Y 314.906,Z 357.352,A -85,B 0,C 180,E1 -16685.382,E2 -16685.382} C_VEL
LIN {X 0,Y 306.072,Z 337.18,A -85,B 0,C 180,E1 -16687.012,E2 -16687.012} C_VEL
LIN {X 0,Y 298.453,Z 321.501,A -85,B 0,C 180,E1 -16688.458,E2 -16688.458} C_VEL
LIN {X 0,Y 294.921,Z 314.403,A -85,B 0,C 180,E1 -16689.173,E2 -16689.173} C_VEL
LIN {X 0,Y 291.333,Z 301.812,A -85,B 0,C 180,E1 -16693.203,E2 -16693.203} C_VEL
LIN {X 0,Y 291.289,Z 301.824,A -85,B 0,C 180,E1 -16697.5,E2 -16697.5} C_VEL
LIN {X 0,Y 291.335,Z 301.813,A -85,B 0,C 180,E1 -16701.153,E2 -16701.153} C_VEL
LIN {X 0,Y 291.356,Z 301.807,A -85,B 0,C 180,E1 -16704.623,E2 -16704.623} C_VEL
LIN {X 0,Y 291.367,Z 301.817,A -85,B 0,C 180,E1 -16707.948,E2 -16707.948} C_VEL
LIN {X 0,Y 291.32,Z 301.822,A -85,B 0,C 180,E1 -16711.15,E2 -16711.15} C_VEL
LIN {X 0,Y 291.343,Z 301.824,A -85,B 0,C 180,E1 -16714.263,E2 -16714.263} C_VEL
LIN {X 0,Y 291.351,Z 301.818,A -85,B 0,C 180,E1 -16717.295,E2 -16717.295} C_VEL
LIN {X 0,Y 291.388,Z 301.81,A -85,B 0,C 180,E1 -16720.263,E2 -16720.263} C_VEL
LIN {X 0,Y 291.497,Z 301.793,A -85,B 0,C 180,E1 -16724.663,E2 -16724.663} C_VEL
LIN {X 0,Y 291.524,Z 301.771,A -85,B 0,C 180,E1 -16728.878,E2 -16728.878} C_VEL
LIN {X 0,Y 291.628,Z 301.784,A -85,B 0,C 180,E1 -16731.684,E2 -16731.684} C_VEL
LIN {X 0,Y 291.589,Z 301.777,A -85,B 0,C 180,E1 -16734.465,E2 -16734.465} C_VEL
LIN {X 0,Y 291.868,Z 301.734,A -85,B 0,C 180,E1 -16738.618,E2 -16738.618} C_VEL
LIN {X 0,Y 291.865,Z 301.754,A -85,B 0,C 180,E1 -16741.377,E2 -16741.377} C_VEL
LIN {X 0,Y 291.663,Z 301.738,A -85,B 0,C 180,E1 -16746.917,E2 -16746.917} C_VEL
LIN {X 0,Y 291.556,Z 301.783,A -85,B 0,C 180,E1 -16749.712,E2 -16749.712} C_VEL
LIN {X 0,Y 291.507,Z 301.787,A -85,B 0,C 180,E1 -16753.948,E2 -16753.948} C_VEL
LIN {X 0,Y 291.424,Z 301.768,A -85,B 0,C 180,E1 -16756.819,E2 -16756.819} C_VEL
LIN {X 0,Y 291.416,Z 301.798,A -85,B 0,C 180,E1 -16759.858,E2 -16759.858} C_VEL
LIN {X 0,Y 291.324,Z 301.812,A -85,B 0,C 180,E1 -16764.209,E2 -16764.209} C_VEL
LIN {X 0,Y 291.318,Z 301.784,A -85,B 0,C 180,E1 -16767.279,E2 -16767.279} C_VEL
LIN {X 0,Y 291.291,Z 301.819,A -85,B 0,C 180,E1 -16770.439,E2 -16770.439} C_VEL
LIN {X 0,Y 291.332,Z 301.813,A -85,B 0,C 180,E1 -16773.696,E2 -16773.696} C_VEL
LIN {X 0,Y 291.34,Z 301.787,A -85,B 0,C 180,E1 -16777.245,E2 -16777.245} C_VEL
LIN {X 0,Y 291.288,Z 301.825,A -85,B 0,C 180,E1 -16780.646,E2 -16780.646} C_VEL
LIN {X 0,Y 291.269,Z 301.806,A -85,B 0,C 180,E1 -16784.402,E2 -16784.402} C_VEL
LIN {X 0,Y 291.313,Z 301.822,A -85,B 0,C 180,E1 -16788.403,E2 -16788.403} C_VEL
LIN {X 0,Y 291.333,Z 301.813,A -85,B 0,C 180,E1 -16791.155,E2 -16791.155} C_VEL
LIN {X 0,Y 291.341,Z 301.81,A -85,B 0,C 180,E1 -16794.624,E2 -16794.624} C_VEL
LIN {X 0,Y 291.351,Z 301.814,A -85,B 0,C 180,E1 -16797.948,E2 -16797.948} C_VEL
LIN {X 0,Y 291.358,Z 301.809,A -85,B 0,C 180,E1 -16801.156,E2 -16801.156} C_VEL
LIN {X 0,Y 291.398,Z 301.802,A -85,B 0,C 180,E1 -16804.27,E2 -16804.27} C_VEL
LIN {X 0,Y 291.359,Z 301.82,A -85,B 0,C 180,E1 -16807.298,E2 -16807.298} C_VEL
LIN {X 0,Y 291.443,Z 301.799,A -85,B 0,C 180,E1 -16810.269,E2 -16810.269} C_VEL
LIN {X 0,Y 291.525,Z 301.794,A -85,B 0,C 180,E1 -16814.633,E2 -16814.633} C_VEL
LIN {X 0,Y 291.522,Z 301.794,A -85,B 0,C 180,E1 -16818.88,E2 -16818.88} C_VEL
LIN {X 0,Y 291.631,Z 301.791,A -85,B 0,C 180,E1 -16820.494,E2 -16820.494} C_VEL
LIN {X 0,Y 292.688,Z 304.704,A -85,B 0,C 180,E1 -16820.737,E2 -16820.737} C_VEL
LIN {X 0,Y 294.253,Z 306.974,A -85,B 0,C 180,E1 -16821.028,E2 -16821.028} C_VEL
LIN {X 0,Y 300.389,Z 317.473,A -85,B 0,C 180,E1 -16822.178,E2 -16822.178} C_VEL
LIN {X 0,Y 310.306,Z 337.373,A -85,B 0,C 180,E1 -16824.01,E2 -16824.01} C_VEL
LIN {X 0,Y 317.226,Z 353.284,A -85,B 0,C 180,E1 -16825.266,E2 -16825.266} C_VEL
LIN {X 0,Y 314.313,Z 430.328,A -85,B 0,C 180,E1 -16827.076,E2 -16827.076} C_VEL
LIN {X 0,Y 312.845,Z 465.996,A -85,B 0,C 180,E1 -16827.948,E2 -16827.948} C_VEL
LIN {X 0,Y 311.616,Z 481.925,A -85,B 0,C 180,E1 -16828.586,E2 -16828.586} C_VEL
LIN {X 0,Y 310.054,Z 496.961,A -85,B 0,C 180,E1 -16829.456,E2 -16829.456} C_VEL
LIN {X 0,Y 308.273,Z 510.587,A -85,B 0,C 180,E1 -16830.489,E2 -16830.489} C_VEL
LIN {X 0,Y 306.12,Z 524.354,A -85,B 0,C 180,E1 -16831.808,E2 -16831.808} C_VEL
LIN {X 0,Y 303.826,Z 537.079,A -85,B 0,C 180,E1 -16833.315,E2 -16833.315} C_VEL
LIN {X 0,Y 301.503,Z 548.851,A -85,B 0,C 180,E1 -16835.014,E2 -16835.014} C_VEL
LIN {X 0,Y 298.974,Z 560.615,A -85,B 0,C 180,E1 -16837.065,E2 -16837.065} C_VEL
LIN {X 0,Y 296.806,Z 570.652,A -85,B 0,C 180,E1 -16839.196,E2 -16839.196} C_VEL
LIN {X 0,Y 294.807,Z 579.425,A -85,B 0,C 180,E1 -16841.433,E2 -16841.433} C_VEL
LIN {X 0,Y 293.054,Z 587.342,A -85,B 0,C 180,E1 -16843.875,E2 -16843.875} C_VEL
LIN {X 0,Y 291.816,Z 593.53,A -85,B 0,C 180,E1 -16846.193,E2 -16846.193} C_VEL
LIN {X 0,Y 290.725,Z 599.253,A -85,B 0,C 180,E1 -16848.842,E2 -16848.842} C_VEL
LIN {X 0,Y 290.098,Z 603.385,A -85,B 0,C 180,E1 -16851.308,E2 -16851.308} C_VEL
LIN {X 0,Y 289.754,Z 605.438,A -85,B 0,C 180,E1 -16852.834,E2 -16852.834} C_VEL
LIN {X 0,Y 289.252,Z 608.509,A -85,B 0,C 180,E1 -16855.981,E2 -16855.981} C_VEL
LIN {X 0,Y 289.067,Z 610.06,A -85,B 0,C 180,E1 -16859.093,E2 -16859.093} C_VEL
LIN {X 0,Y 289.12,Z 610.223,A -85,B 0,C 180,E1 -16861.709,E2 -16861.709} C_VEL
LIN {X 0,Y 289.318,Z 609.419,A -85,B 0,C 180,E1 -16864.324,E2 -16864.324} C_VEL
LIN {X 0,Y 289.773,Z 607.247,A -85,B 0,C 180,E1 -16867.323,E2 -16867.323} C_VEL
LIN {X 0,Y 290.534,Z 604.258,A -85,B 0,C 180,E1 -16869.92,E2 -16869.92} C_VEL
LIN {X 0,Y 291.464,Z 600.221,A -85,B 0,C 180,E1 -16872.464,E2 -16872.464} C_VEL
LIN {X 0,Y 292.79,Z 594.902,A -85,B 0,C 180,E1 -16875.079,E2 -16875.079} C_VEL
LIN {X 0,Y 294.587,Z 588.216,A -85,B 0,C 180,E1 -16877.693,E2 -16877.693} C_VEL
LIN {X 0,Y 296.863,Z 580.014,A -85,B 0,C 180,E1 -16880.271,E2 -16880.271} C_VEL
LIN {X 0,Y 299.311,Z 571.191,A -85,B 0,C 180,E1 -16882.542,E2 -16882.542} C_VEL
LIN {X 0,Y 302.215,Z 560.637,A -85,B 0,C 180,E1 -16884.766,E2 -16884.766} C_VEL
LIN {X 0,Y 304.91,Z 550.103,A -85,B 0,C 180,E1 -16886.609,E2 -16886.609} C_VEL
LIN {X 0,Y 307.748,Z 538.254,A -85,B 0,C 180,E1 -16888.318,E2 -16888.318} C_VEL
LIN {X 0,Y 310.492,Z 525.166,A -85,B 0,C 180,E1 -16889.873,E2 -16889.873} C_VEL
LIN {X 0,Y 313.144,Z 510.739,A -85,B 0,C 180,E1 -16891.234,E2 -16891.234} C_VEL
LIN {X 0,Y 313.449,Z 505.478,A -85,B 0,C 180,E1 -16891.729,E2 -16891.729} C_VEL
LIN {X 0,Y 312.394,Z 496.969,A -85,B 0,C 180,E1 -16892.647,E2 -16892.647} C_VEL
LIN {X 0,Y 311.232,Z 488.279,A -85,B 0,C 180,E1 -16893.486,E2 -16893.486} C_VEL
LIN {X 0,Y 311.339,Z 482.743,A -85,B 0,C 180,E1 -16893.85,E2 -16893.85} C_VEL
LIN {X 0,Y 312.804,Z 467.094,A -85,B 0,C 180,E1 -16894.471,E2 -16894.471} C_VEL
LIN {X 0,Y 318.024,Z 360.191,A -85,B 0,C 180,E1 -16897.091,E2 -16897.091} C_VEL
LIN {X 0,Y 312.453,Z 348.108,A -85,B 0,C 180,E1 -16898.413,E2 -16898.413} C_VEL
LIN {X 0,Y 305.374,Z 334.832,A -85,B 0,C 180,E1 -16900.168,E2 -16900.168} C_VEL
LIN {X 0,Y 299.737,Z 325.52,A -85,B 0,C 180,E1 -16901.638,E2 -16901.638} C_VEL
LIN {X 0,Y 294.47,Z 317.287,A -85,B 0,C 180,E1 -16903.104,E2 -16903.104} C_VEL
LIN {X 0,Y 290.909,Z 312.315,A -85,B 0,C 180,E1 -16904.139,E2 -16904.139} C_VEL
LIN {X 0,Y 288.564,Z 309.164,A -85,B 0,C 180,E1 -16904.851,E2 -16904.851} C_VEL
LIN {X 0,Y 287.962,Z 307.934,A -85,B 0,C 180,E1 -16905.057,E2 -16905.057} C_VEL
LIN {X 0,Y 285.627,Z 305.746,A -85,B 0,C 180,E1 -16905.758,E2 -16905.758} C_VEL
LIN {X 0,Y 284.534,Z 303.081,A -85,B 0,C 180,E1 -16906.204,E2 -16906.204} C_VEL
LIN {X 0,Y 284.463,Z 302.677,A -85,B 0,C 180,E1 -16906.428,E2 -16906.428} C_VEL
LIN {X 0,Y 284.616,Z 302.655,A -85,B 0,C 180,E1 -16910.999,E2 -16910.999} C_VEL
LIN {X 0,Y 284.586,Z 302.657,A -85,B 0,C 180,E1 -16914.333,E2 -16914.333} C_VEL
LIN {X 0,Y 284.845,Z 302.625,A -85,B 0,C 180,E1 -16918.589,E2 -16918.589} C_VEL
LIN {X 0,Y 284.845,Z 302.624,A -85,B 0,C 180,E1 -16921.416,E2 -16921.416} C_VEL
LIN {X 0,Y 284.645,Z 302.65,A -85,B 0,C 180,E1 -16927.094,E2 -16927.094} C_VEL
LIN {X 0,Y 284.507,Z 302.67,A -85,B 0,C 180,E1 -16929.96,E2 -16929.96} C_VEL
LIN {X 0,Y 284.456,Z 302.67,A -85,B 0,C 180,E1 -16934.306,E2 -16934.306} C_VEL
LIN {X 0,Y 284.326,Z 302.694,A -85,B 0,C 180,E1 -16938.746,E2 -16938.746} C_VEL
LIN {X 0,Y 284.305,Z 302.689,A -85,B 0,C 180,E1 -16943.3,E2 -16943.3} C_VEL
LIN {X 0,Y 284.282,Z 302.697,A -85,B 0,C 180,E1 -16947.132,E2 -16947.132} C_VEL
LIN {X 0,Y 284.269,Z 302.698,A -85,B 0,C 180,E1 -16950.086,E2 -16950.086} C_VEL
LIN {X 0,Y 284.301,Z 302.695,A -85,B 0,C 180,E1 -16952.948,E2 -16952.948} C_VEL
LIN {X 0,Y 284.315,Z 302.688,A -85,B 0,C 180,E1 -16956.391,E2 -16956.391} C_VEL
LIN {X 0,Y 284.266,Z 302.705,A -85,B 0,C 180,E1 -16960.119,E2 -16960.119} C_VEL
LIN {X 0,Y 287.187,Z 311.357,A -85,B 0,C 180,E1 -16964.292,E2 -16964.292} C_VEL
LIN {X 0,Y 287.666,Z 312.47,A -85,B 0,C 180,E1 -16964.695,E2 -16964.695} C_VEL
LIN {X 0,Y 290.89,Z 317.296,A -85,B 0,C 180,E1 -16965.693,E2 -16965.693} C_VEL
LIN {X 0,Y 295.78,Z 325.083,A -85,B 0,C 180,E1 -16967.13,E2 -16967.13} C_VEL
LIN {X 0,Y 301.079,Z 333.82,A -85,B 0,C 180,E1 -16968.582,E2 -16968.582} C_VEL
LIN {X 0,Y 307.921,Z 346.597,A -85,B 0,C 180,E1 -16970.356,E2 -16970.356} C_VEL
LIN {X 0,Y 314.896,Z 361.598,A -85,B 0,C 180,E1 -16972.077,E2 -16972.077} C_VEL
LIN {X 0,Y 317.029,Z 367.131,A -85,B 0,C 180,E1 -16972.604,E2 -16972.604} C_VEL
LIN {X 0,Y 317.648,Z 372.698,A -85,B 0,C 180,E1 -16972.881,E2 -16972.881} C_VEL
LIN {X 0,Y 312.37,Z 479.892,A -85,B 0,C 180,E1 -16975.482,E2 -16975.482} C_VEL
LIN {X 0,Y 310.736,Z 496.248,A -85,B 0,C 180,E1 -16976.108,E2 -16976.108} C_VEL
LIN {X 0,Y 308.537,Z 511.662,A -85,B 0,C 180,E1 -16976.959,E2 -16976.959} C_VEL
LIN {X 0,Y 306.297,Z 525.091,A -85,B 0,C 180,E1 -16977.955,E2 -16977.955} C_VEL
LIN {X 0,Y 303.592,Z 538.497,A -85,B 0,C 180,E1 -16979.21,E2 -16979.21} C_VEL
LIN {X 0,Y 300.533,Z 551.945,A -85,B 0,C 180,E1 -16980.781,E2 -16980.781} C_VEL
LIN {X 0,Y 297.389,Z 564.311,A -85,B 0,C 180,E1 -16982.561,E2 -16982.561} C_VEL
LIN {X 0,Y 294.337,Z 575.617,A -85,B 0,C 180,E1 -16984.547,E2 -16984.547} C_VEL
LIN {X 0,Y 291.587,Z 585.728,A -85,B 0,C 180,E1 -16986.703,E2 -16986.703} C_VEL
LIN {X 0,Y 289.037,Z 594.629,A -85,B 0,C 180,E1 -16988.984,E2 -16988.984} C_VEL
LIN {X 0,Y 286.88,Z 602.517,A -85,B 0,C 180,E1 -16991.43,E2 -16991.43} C_VEL
LIN {X 0,Y 284.942,Z 609.909,A -85,B 0,C 180,E1 -16994.259,E2 -16994.259} C_VEL
LIN {X 0,Y 283.657,Z 615.793,A -85,B 0,C 180,E1 -16997.116,E2 -16997.116} C_VEL
LIN {X 0,Y 282.794,Z 620.331,A -85,B 0,C 180,E1 -16999.982,E2 -16999.982} C_VEL
LIN {X 0,Y 282.375,Z 623.615,A -85,B 0,C 180,E1 -17002.852,E2 -17002.852} C_VEL
LIN {X 0,Y 282.271,Z 625.652,A -85,B 0,C 180,E1 -17005.717,E2 -17005.717} C_VEL
LIN {X 0,Y 282.336,Z 626.512,A -85,B 0,C 180,E1 -17008.574,E2 -17008.574} C_VEL
LIN {X 0,Y 282.337,Z 626.212,A -85,B 0,C 180,E1 -17011.427,E2 -17011.427} C_VEL
LIN {X 0,Y 282.29,Z 624.736,A -85,B 0,C 180,E1 -17014.284,E2 -17014.284} C_VEL
LIN {X 0,Y 282.398,Z 622.054,A -85,B 0,C 180,E1 -17017.149,E2 -17017.149} C_VEL
LIN {X 0,Y 282.767,Z 618.076,A -85,B 0,C 180,E1 -17020.02,E2 -17020.02} C_VEL
LIN {X 0,Y 283.57,Z 612.712,A -85,B 0,C 180,E1 -17022.889,E2 -17022.889} C_VEL
LIN {X 0,Y 284.735,Z 605.841,A -85,B 0,C 180,E1 -17025.754,E2 -17025.754} C_VEL
LIN {X 0,Y 286.534,Z 597.279,A -85,B 0,C 180,E1 -17028.594,E2 -17028.594} C_VEL
LIN {X 0,Y 288.643,Z 588.121,A -85,B 0,C 180,E1 -17031.047,E2 -17031.047} C_VEL
LIN {X 0,Y 290.847,Z 577.823,A -85,B 0,C 180,E1 -17033.328,E2 -17033.328} C_VEL
LIN {X 0,Y 293.105,Z 567.671,A -85,B 0,C 180,E1 -17035.189,E2 -17035.189} C_VEL
LIN {X 0,Y 295.801,Z 555.582,A -85,B 0,C 180,E1 -17037.026,E2 -17037.026} C_VEL
LIN {X 0,Y 298.364,Z 542.312,A -85,B 0,C 180,E1 -17038.681,E2 -17038.681} C_VEL
LIN {X 0,Y 300.806,Z 528.413,A -85,B 0,C 180,E1 -17040.068,E2 -17040.068} C_VEL
LIN {X 0,Y 302.871,Z 514.297,A -85,B 0,C 180,E1 -17041.181,E2 -17041.181} C_VEL
LIN {X 0,Y 304.721,Z 499.853,A -85,B 0,C 180,E1 -17042.037,E2 -17042.037} C_VEL
LIN {X 0,Y 306.153,Z 484.27,A -85,B 0,C 180,E1 -17042.696,E2 -17042.696} C_VEL
LIN {X 0,Y 307.166,Z 463.293,A -85,B 0,C 180,E1 -17043.258,E2 -17043.258} C_VEL
LIN {X 0,Y 310.885,Z 370.157,A -85,B 0,C 180,E1 -17045.481,E2 -17045.481} C_VEL
LIN {X 0,Y 309.124,Z 360.086,A -85,B 0,C 180,E1 -17045.976,E2 -17045.976} C_VEL
LIN {X 0,Y 300.531,Z 340.377,A -85,B 0,C 180,E1 -17047.608,E2 -17047.608} C_VEL
LIN {X 0,Y 293.322,Z 325.416,A -85,B 0,C 180,E1 -17049.029,E2 -17049.029} C_VEL
LIN {X 0,Y 287.517,Z 314.076,A -85,B 0,C 180,E1 -17050.249,E2 -17050.249} C_VEL
LIN {X 0,Y 284.985,Z 305.122,A -85,B 0,C 180,E1 -17053.19,E2 -17053.19} C_VEL
LIN {X 0,Y 284.241,Z 302.698,A -85,B 0,C 180,E1 -17054.057,E2 -17054.057} C_VEL
LIN {X 0,Y 284.241,Z 302.708,A -85,B 0,C 180,E1 -17058.117,E2 -17058.117} C_VEL
LIN {X 0,Y 284.297,Z 302.695,A -85,B 0,C 180,E1 -17061.827,E2 -17061.827} C_VEL
LIN {X 0,Y 284.309,Z 302.68,A -85,B 0,C 180,E1 -17065.349,E2 -17065.349} C_VEL
LIN {X 0,Y 284.28,Z 302.698,A -85,B 0,C 180,E1 -17068.722,E2 -17068.722} C_VEL
LIN {X 0,Y 284.264,Z 302.7,A -85,B 0,C 180,E1 -17071.98,E2 -17071.98} C_VEL
LIN {X 0,Y 284.284,Z 302.702,A -85,B 0,C 180,E1 -17075.146,E2 -17075.146} C_VEL
LIN {X 0,Y 284.3,Z 302.703,A -85,B 0,C 180,E1 -17078.233,E2 -17078.233} C_VEL
LIN {X 0,Y 284.331,Z 302.691,A -85,B 0,C 180,E1 -17081.255,E2 -17081.255} C_VEL
LIN {X 0,Y 284.461,Z 302.652,A -85,B 0,C 180,E1 -17085.694,E2 -17085.694} C_VEL
LIN {X 0,Y 284.509,Z 302.658,A -85,B 0,C 180,E1 -17090.04,E2 -17090.04} C_VEL
LIN {X 0,Y 284.632,Z 302.654,A -85,B 0,C 180,E1 -17092.906,E2 -17092.906} C_VEL
LIN {X 0,Y 284.834,Z 302.608,A -85,B 0,C 180,E1 -17098.584,E2 -17098.584} C_VEL
LIN {X 0,Y 284.832,Z 302.631,A -85,B 0,C 180,E1 -17101.412,E2 -17101.412} C_VEL
LIN {X 0,Y 284.619,Z 302.615,A -85,B 0,C 180,E1 -17107.09,E2 -17107.09} C_VEL
LIN {X 0,Y 284.504,Z 302.664,A -85,B 0,C 180,E1 -17109.955,E2 -17109.955} C_VEL
LIN {X 0,Y 284.456,Z 302.664,A -85,B 0,C 180,E1 -17114.301,E2 -17114.301} C_VEL
LIN {X 0,Y 284.354,Z 302.665,A -85,B 0,C 180,E1 -17118.739,E2 -17118.739} C_VEL
LIN {X 0,Y 284.294,Z 302.697,A -85,B 0,C 180,E1 -17121.763,E2 -17121.763} C_VEL
LIN {X 0,Y 284.278,Z 302.68,A -85,B 0,C 180,E1 -17124.849,E2 -17124.849} C_VEL
LIN {X 0,Y 284.249,Z 302.668,A -85,B 0,C 180,E1 -17128.016,E2 -17128.016} C_VEL
LIN {X 0,Y 284.267,Z 302.699,A -85,B 0,C 180,E1 -17131.274,E2 -17131.274} C_VEL
LIN {X 0,Y 284.325,Z 302.667,A -85,B 0,C 180,E1 -17135.344,E2 -17135.344} C_VEL
LIN {X 0,Y 284.283,Z 302.675,A -85,B 0,C 180,E1 -17138.17,E2 -17138.17} C_VEL
LIN {X 0,Y 284.224,Z 302.705,A -85,B 0,C 180,E1 -17142.115,E2 -17142.115} C_VEL
LIN {X 0,Y 284.242,Z 302.68,A -85,B 0,C 180,E1 -17146.187,E2 -17146.187} C_VEL
LIN {X 0,Y 284.293,Z 302.699,A -85,B 0,C 180,E1 -17150.022,E2 -17150.022} C_VEL
LIN {X 0,Y 284.309,Z 302.676,A -85,B 0,C 180,E1 -17153.611,E2 -17153.611} C_VEL
LIN {X 0,Y 284.292,Z 302.697,A -85,B 0,C 180,E1 -17157.189,E2 -17157.189} C_VEL
LIN {X 0,Y 284.336,Z 302.676,A -85,B 0,C 180,E1 -17160.374,E2 -17160.374} C_VEL
LIN {X 0,Y 284.361,Z 302.684,A -85,B 0,C 180,E1 -17163.585,E2 -17163.585} C_VEL
LIN {X 0,Y 284.318,Z 302.693,A -85,B 0,C 180,E1 -17166.703,E2 -17166.703} C_VEL
LIN {X 0,Y 284.384,Z 302.689,A -85,B 0,C 180,E1 -17171.26,E2 -17171.26} C_VEL
LIN {X 0,Y 284.462,Z 302.672,A -85,B 0,C 180,E1 -17174.469,E2 -17174.469} C_VEL
LIN {X 0,Y 284.474,Z 302.674,A -85,B 0,C 180,E1 -17178.601,E2 -17178.601} C_VEL
LIN {X 0,Y 284.501,Z 302.665,A -85,B 0,C 180,E1 -17179.457,E2 -17179.457} C_VEL
LIN {X 0,Y 285.57,Z 305.604,A -85,B 0,C 180,E1 -17179.735,E2 -17179.735} C_VEL
LIN {X 0,Y 287.246,Z 307.945,A -85,B 0,C 180,E1 -17180.057,E2 -17180.057} C_VEL
LIN {X 0,Y 294.904,Z 320.723,A -85,B 0,C 180,E1 -17181.548,E2 -17181.548} C_VEL
LIN {X 0,Y 305.295,Z 341.752,A -85,B 0,C 180,E1 -17183.529,E2 -17183.529} C_VEL
LIN {X 0,Y 311.168,Z 355.339,A -85,B 0,C 180,E1 -17184.628,E2 -17184.628} C_VEL
LIN {X 0,Y 306.711,Z 465.631,A -85,B 0,C 180,E1 -17187.291,E2 -17187.291} C_VEL
LIN {X 0,Y 305.427,Z 481.763,A -85,B 0,C 180,E1 -17187.939,E2 -17187.939} C_VEL
LIN {X 0,Y 303.854,Z 496.61,A -85,B 0,C 180,E1 -17188.805,E2 -17188.805} C_VEL
LIN {X 0,Y 301.973,Z 510.43,A -85,B 0,C 180,E1 -17189.861,E2 -17189.861} C_VEL
LIN {X 0,Y 299.825,Z 523.964,A -85,B 0,C 180,E1 -17191.175,E2 -17191.175} C_VEL
LIN {X 0,Y 297.394,Z 536.811,A -85,B 0,C 180,E1 -17192.708,E2 -17192.708} C_VEL
LIN {X 0,Y 294.991,Z 548.655,A -85,B 0,C 180,E1 -17194.44,E2 -17194.44} C_VEL
LIN {X 0,Y 292.334,Z 560.613,A -85,B 0,C 180,E1 -17196.556,E2 -17196.556} C_VEL
LIN {X 0,Y 290.088,Z 570.582,A -85,B 0,C 180,E1 -17198.708,E2 -17198.708} C_VEL
LIN {X 0,Y 288.102,Z 579.051,A -85,B 0,C 180,E1 -17200.897,E2 -17200.897} C_VEL
LIN {X 0,Y 286.185,Z 587.354,A -85,B 0,C 180,E1 -17203.49,E2 -17203.49} C_VEL
LIN {X 0,Y 284.867,Z 593.491,A -85,B 0,C 180,E1 -17205.822,E2 -17205.822} C_VEL
LIN {X 0,Y 283.649,Z 599.715,A -85,B 0,C 180,E1 -17208.789,E2 -17208.789} C_VEL
LIN {X 0,Y 282.876,Z 604.561,A -85,B 0,C 180,E1 -17211.879,E2 -17211.879} C_VEL
LIN {X 0,Y 282.522,Z 606.45,A -85,B 0,C 180,E1 -17213.453,E2 -17213.453} C_VEL
LIN {X 0,Y 282.088,Z 609.146,A -85,B 0,C 180,E1 -17216.643,E2 -17216.643} C_VEL
LIN {X 0,Y 281.986,Z 610.306,A -85,B 0,C 180,E1 -17219.278,E2 -17219.278} C_VEL
LIN {X 0,Y 282.035,Z 610.405,A -85,B 0,C 180,E1 -17222.093,E2 -17222.093} C_VEL
LIN {X 0,Y 282.28,Z 609.397,A -85,B 0,C 180,E1 -17224.933,E2 -17224.933} C_VEL
LIN {X 0,Y 282.672,Z 607.74,A -85,B 0,C 180,E1 -17227.293,E2 -17227.293} C_VEL
LIN {X 0,Y 283.499,Z 604.603,A -85,B 0,C 180,E1 -17230.13,E2 -17230.13} C_VEL
LIN {X 0,Y 284.551,Z 600.452,A -85,B 0,C 180,E1 -17232.838,E2 -17232.838} C_VEL
LIN {X 0,Y 285.933,Z 595.269,A -85,B 0,C 180,E1 -17235.461,E2 -17235.461} C_VEL
LIN {X 0,Y 287.755,Z 588.833,A -85,B 0,C 180,E1 -17238.061,E2 -17238.061} C_VEL
LIN {X 0,Y 290.237,Z 580.385,A -85,B 0,C 180,E1 -17240.791,E2 -17240.791} C_VEL
LIN {X 0,Y 292.853,Z 571.46,A -85,B 0,C 180,E1 -17243.137,E2 -17243.137} C_VEL
LIN {X 0,Y 296.009,Z 560.464,A -85,B 0,C 180,E1 -17245.49,E2 -17245.49} C_VEL
LIN {X 0,Y 298.901,Z 549.723,A -85,B 0,C 180,E1 -17247.385,E2 -17247.385} C_VEL
LIN {X 0,Y 301.996,Z 537.139,A -85,B 0,C 180,E1 -17249.207,E2 -17249.207} C_VEL
LIN {X 0,Y 304.955,Z 523.62,A -85,B 0,C 180,E1 -17250.79,E2 -17250.79} C_VEL
LIN {X 0,Y 307.497,Z 510.054,A -85,B 0,C 180,E1 -17252.065,E2 -17252.065} C_VEL
LIN {X 0,Y 309.725,Z 495.835,A -85,B 0,C 180,E1 -17253.11,E2 -17253.11} C_VEL
LIN {X 0,Y 311.339,Z 482.743,A -85,B 0,C 180,E1 -17253.85,E2 -17253.85} C_VEL
LIN {X 0,Y 311.468,Z 477.124,A -85,B 0,C 180,E1 -17254.185,E2 -17254.185} C_VEL
LIN {X 0,Y 308.582,Z 460.668,A -85,B 0,C 180,E1 -17255.35,E2 -17255.35} C_VEL
LIN {X 0,Y 308.08,Z 454.959,A -85,B 0,C 180,E1 -17255.62,E2 -17255.62} C_VEL
LIN {X 0,Y 308.111,Z 453.014,A -85,B 0,C 180,E1 -17255.677,E2 -17255.677} C_VEL
LIN {X 0,Y 312.633,Z 362.515,A -85,B 0,C 180,E1 -17257.901,E2 -17257.901} C_VEL
LIN {X 0,Y 307.644,Z 351.704,A -85,B 0,C 180,E1 -17259.148,E2 -17259.148} C_VEL
LIN {X 0,Y 301.134,Z 339.335,A -85,B 0,C 180,E1 -17260.83,E2 -17260.83} C_VEL
LIN {X 0,Y 294.278,Z 327.828,A -85,B 0,C 180,E1 -17262.723,E2 -17262.723} C_VEL
LIN {X 0,Y 290.389,Z 321.888,A -85,B 0,C 180,E1 -17263.863,E2 -17263.863} C_VEL
LIN {X 0,Y 287.427,Z 317.763,A -85,B 0,C 180,E1 -17264.763,E2 -17264.763} C_VEL
LIN {X 0,Y 284.369,Z 313.539,A -85,B 0,C 180,E1 -17265.74,E2 -17265.74} C_VEL
LIN {X 0,Y 282.011,Z 310.674,A -85,B 0,C 180,E1 -17266.51,E2 -17266.51} C_VEL
LIN {X 0,Y 280.948,Z 308.82,A -85,B 0,C 180,E1 -17266.9,E2 -17266.9} C_VEL
LIN {X 0,Y 278.663,Z 306.772,A -85,B 0,C 180,E1 -17267.67,E2 -17267.67} C_VEL
LIN {X 0,Y 277.552,Z 304.287,A -85,B 0,C 180,E1 -17268.13,E2 -17268.13} C_VEL
LIN {X 0,Y 277.434,Z 303.554,A -85,B 0,C 180,E1 -17268.218,E2 -17268.218} C_VEL
LIN {X 0,Y 277.588,Z 303.529,A -85,B 0,C 180,E1 -17271.265,E2 -17271.265} C_VEL
LIN {X 0,Y 277.557,Z 303.532,A -85,B 0,C 180,E1 -17274.189,E2 -17274.189} C_VEL
LIN {X 0,Y 277.811,Z 303.501,A -85,B 0,C 180,E1 -17278.553,E2 -17278.553} C_VEL
LIN {X 0,Y 277.811,Z 303.5,A -85,B 0,C 180,E1 -17281.452,E2 -17281.452} C_VEL
LIN {X 0,Y 277.602,Z 303.525,A -85,B 0,C 180,E1 -17287.274,E2 -17287.274} C_VEL
LIN {X 0,Y 277.448,Z 303.546,A -85,B 0,C 180,E1 -17290.216,E2 -17290.216} C_VEL
LIN {X 0,Y 277.403,Z 303.55,A -85,B 0,C 180,E1 -17294.678,E2 -17294.678} C_VEL
LIN {X 0,Y 277.279,Z 303.569,A -85,B 0,C 180,E1 -17299.241,E2 -17299.241} C_VEL
LIN {X 0,Y 277.255,Z 303.57,A -85,B 0,C 180,E1 -17303.929,E2 -17303.929} C_VEL
LIN {X 0,Y 277.232,Z 303.576,A -85,B 0,C 180,E1 -17307.471,E2 -17307.471} C_VEL
LIN {X 0,Y 277.225,Z 303.576,A -85,B 0,C 180,E1 -17310.468,E2 -17310.468} C_VEL
LIN {X 0,Y 277.243,Z 303.568,A -85,B 0,C 180,E1 -17313.898,E2 -17313.898} C_VEL
LIN {X 0,Y 277.248,Z 303.57,A -85,B 0,C 180,E1 -17317.475,E2 -17317.475} C_VEL
LIN {X 0,Y 277.254,Z 303.725,A -85,B 0,C 180,E1 -17318.393,E2 -17318.393} C_VEL
LIN {X 0,Y 280.026,Z 311.705,A -85,B 0,C 180,E1 -17322.6,E2 -17322.6} C_VEL
LIN {X 0,Y 283.888,Z 317.397,A -85,B 0,C 180,E1 -17323.935,E2 -17323.935} C_VEL
LIN {X 0,Y 288.735,Z 324.82,A -85,B 0,C 180,E1 -17325.492,E2 -17325.492} C_VEL
LIN {X 0,Y 292.361,Z 330.727,A -85,B 0,C 180,E1 -17326.589,E2 -17326.589} C_VEL
LIN {X 0,Y 297.31,Z 339.071,A -85,B 0,C 180,E1 -17328.002,E2 -17328.002} C_VEL
LIN {X 0,Y 303.618,Z 351.045,A -85,B 0,C 180,E1 -17329.709,E2 -17329.709} C_VEL
LIN {X 0,Y 310.418,Z 366.052,A -85,B 0,C 180,E1 -17331.47,E2 -17331.47} C_VEL
LIN {X 0,Y 311.953,Z 370.301,A -85,B 0,C 180,E1 -17331.873,E2 -17331.873} C_VEL
LIN {X 0,Y 312.32,Z 373.534,A -85,B 0,C 180,E1 -17332.041,E2 -17332.041} C_VEL
LIN {X 0,Y 306.83,Z 480.025,A -85,B 0,C 180,E1 -17334.667,E2 -17334.667} C_VEL
LIN {X 0,Y 305.243,Z 495.443,A -85,B 0,C 180,E1 -17335.262,E2 -17335.262} C_VEL
LIN {X 0,Y 303.036,Z 510.407,A -85,B 0,C 180,E1 -17336.08,E2 -17336.08} C_VEL
LIN {X 0,Y 300.692,Z 523.951,A -85,B 0,C 180,E1 -17337.085,E2 -17337.085} C_VEL
LIN {X 0,Y 297.793,Z 537.944,A -85,B 0,C 180,E1 -17338.397,E2 -17338.397} C_VEL
LIN {X 0,Y 294.663,Z 551.117,A -85,B 0,C 180,E1 -17339.944,E2 -17339.944} C_VEL
LIN {X 0,Y 291.406,Z 563.587,A -85,B 0,C 180,E1 -17341.752,E2 -17341.752} C_VEL
LIN {X 0,Y 288.383,Z 574.083,A -85,B 0,C 180,E1 -17343.593,E2 -17343.593} C_VEL
LIN {X 0,Y 285.419,Z 584.435,A -85,B 0,C 180,E1 -17345.796,E2 -17345.796} C_VEL
LIN {X 0,Y 282.792,Z 593.457,A -85,B 0,C 180,E1 -17348.114,E2 -17348.114} C_VEL
LIN {X 0,Y 280.384,Z 601.517,A -85,B 0,C 180,E1 -17350.604,E2 -17350.604} C_VEL
LIN {X 0,Y 278.483,Z 608.241,A -85,B 0,C 180,E1 -17353.13,E2 -17353.13} C_VEL
LIN {X 0,Y 276.999,Z 614.435,A -85,B 0,C 180,E1 -17356.053,E2 -17356.053} C_VEL
LIN {X 0,Y 275.921,Z 619.229,A -85,B 0,C 180,E1 -17358.988,E2 -17358.988} C_VEL
LIN {X 0,Y 275.484,Z 621.997,A -85,B 0,C 180,E1 -17361.196,E2 -17361.196} C_VEL
LIN {X 0,Y 275.213,Z 624.634,A -85,B 0,C 180,E1 -17364.138,E2 -17364.138} C_VEL
LIN {X 0,Y 275.231,Z 626.046,A -85,B 0,C 180,E1 -17367.073,E2 -17367.073} C_VEL
LIN {X 0,Y 275.28,Z 626.296,A -85,B 0,C 180,E1 -17370.001,E2 -17370.001} C_VEL
LIN {X 0,Y 275.236,Z 625.377,A -85,B 0,C 180,E1 -17372.928,E2 -17372.928} C_VEL
LIN {X 0,Y 275.242,Z 623.267,A -85,B 0,C 180,E1 -17375.863,E2 -17375.863} C_VEL
LIN {X 0,Y 275.502,Z 619.921,A -85,B 0,C 180,E1 -17378.805,E2 -17378.805} C_VEL
LIN {X 0,Y 276.042,Z 615.227,A -85,B 0,C 180,E1 -17381.753,E2 -17381.753} C_VEL
LIN {X 0,Y 277.149,Z 609.09,A -85,B 0,C 180,E1 -17384.69,E2 -17384.69} C_VEL
LIN {X 0,Y 278.734,Z 601.356,A -85,B 0,C 180,E1 -17387.612,E2 -17387.612} C_VEL
LIN {X 0,Y 280.541,Z 593.045,A -85,B 0,C 180,E1 -17390.149,E2 -17390.149} C_VEL
LIN {X 0,Y 282.699,Z 584.59,A -85,B 0,C 180,E1 -17392.279,E2 -17392.279} C_VEL
LIN {X 0,Y 284.934,Z 574.487,A -85,B 0,C 180,E1 -17394.435,E2 -17394.435} C_VEL
LIN {X 0,Y 287.294,Z 563.895,A -85,B 0,C 180,E1 -17396.32,E2 -17396.32} C_VEL
LIN {X 0,Y 289.873,Z 552.367,A -85,B 0,C 180,E1 -17398.018,E2 -17398.018} C_VEL
LIN {X 0,Y 292.625,Z 538.389,A -85,B 0,C 180,E1 -17399.693,E2 -17399.693} C_VEL
LIN {X 0,Y 295.074,Z 524.473,A -85,B 0,C 180,E1 -17401.018,E2 -17401.018} C_VEL
LIN {X 0,Y 297.149,Z 510.657,A -85,B 0,C 180,E1 -17402.051,E2 -17402.051} C_VEL
LIN {X 0,Y 298.944,Z 495.827,A -85,B 0,C 180,E1 -17402.882,E2 -17402.882} C_VEL
LIN {X 0,Y 300.255,Z 480.726,A -85,B 0,C 180,E1 -17403.471,E2 -17403.471} C_VEL
LIN {X 0,Y 304.829,Z 371.175,A -85,B 0,C 180,E1 -17406.163,E2 -17406.163} C_VEL
LIN {X 0,Y 303.351,Z 362.707,A -85,B 0,C 180,E1 -17406.59,E2 -17406.59} C_VEL
LIN {X 0,Y 294.697,Z 342.825,A -85,B 0,C 180,E1 -17408.297,E2 -17408.297} C_VEL
LIN {X 0,Y 286.39,Z 325.774,A -85,B 0,C 180,E1 -17409.992,E2 -17409.992} C_VEL
LIN {X 0,Y 280.202,Z 313.904,A -85,B 0,C 180,E1 -17411.33,E2 -17411.33} C_VEL
LIN {X 0,Y 277.603,Z 305.177,A -85,B 0,C 180,E1 -17414.338,E2 -17414.338} C_VEL
LIN {X 0,Y 277.175,Z 303.587,A -85,B 0,C 180,E1 -17414.913,E2 -17414.913} C_VEL
LIN {X 0,Y 277.186,Z 303.59,A -85,B 0,C 180,E1 -17418.757,E2 -17418.757} C_VEL
LIN {X 0,Y 277.254,Z 303.581,A -85,B 0,C 180,E1 -17422.526,E2 -17422.526} C_VEL
LIN {X 0,Y 277.248,Z 303.56,A -85,B 0,C 180,E1 -17426.102,E2 -17426.102} C_VEL
LIN {X 0,Y 277.23,Z 303.573,A -85,B 0,C 180,E1 -17429.533,E2 -17429.533} C_VEL
LIN {X 0,Y 277.254,Z 303.569,A -85,B 0,C 180,E1 -17432.851,E2 -17432.851} C_VEL
LIN {X 0,Y 277.255,Z 303.572,A -85,B 0,C 180,E1 -17436.071,E2 -17436.071} C_VEL
LIN {X 0,Y 277.284,Z 303.567,A -85,B 0,C 180,E1 -17440.76,E2 -17440.76} C_VEL
LIN {X 0,Y 277.407,Z 303.534,A -85,B 0,C 180,E1 -17445.322,E2 -17445.322} C_VEL
LIN {X 0,Y 277.451,Z 303.533,A -85,B 0,C 180,E1 -17449.784,E2 -17449.784} C_VEL
LIN {X 0,Y 277.588,Z 303.531,A -85,B 0,C 180,E1 -17452.725,E2 -17452.725} C_VEL
LIN {X 0,Y 277.799,Z 303.483,A -85,B 0,C 180,E1 -17458.548,E2 -17458.548} C_VEL
LIN {X 0,Y 277.799,Z 303.507,A -85,B 0,C 180,E1 -17461.447,E2 -17461.447} C_VEL
LIN {X 0,Y 277.576,Z 303.492,A -85,B 0,C 180,E1 -17467.27,E2 -17467.27} C_VEL
LIN {X 0,Y 277.449,Z 303.546,A -85,B 0,C 180,E1 -17470.211,E2 -17470.211} C_VEL
LIN {X 0,Y 277.402,Z 303.534,A -85,B 0,C 180,E1 -17474.673,E2 -17474.673} C_VEL
LIN {X 0,Y 277.309,Z 303.546,A -85,B 0,C 180,E1 -17479.233,E2 -17479.233} C_VEL
LIN {X 0,Y 277.251,Z 303.566,A -85,B 0,C 180,E1 -17483.925,E2 -17483.925} C_VEL
LIN {X 0,Y 277.225,Z 303.538,A -85,B 0,C 180,E1 -17487.466,E2 -17487.466} C_VEL
LIN {X 0,Y 277.218,Z 303.572,A -85,B 0,C 180,E1 -17490.463,E2 -17490.463} C_VEL
LIN {X 0,Y 277.235,Z 303.568,A -85,B 0,C 180,E1 -17493.894,E2 -17493.894} C_VEL
LIN {X 0,Y 277.238,Z 303.543,A -85,B 0,C 180,E1 -17497.47,E2 -17497.47} C_VEL
LIN {X 0,Y 277.172,Z 303.587,A -85,B 0,C 180,E1 -17501.239,E2 -17501.239} C_VEL
LIN {X 0,Y 277.185,Z 303.555,A -85,B 0,C 180,E1 -17505.225,E2 -17505.225} C_VEL
LIN {X 0,Y 277.21,Z 303.582,A -85,B 0,C 180,E1 -17509.51,E2 -17509.51} C_VEL
LIN {X 0,Y 277.244,Z 303.555,A -85,B 0,C 180,E1 -17512.527,E2 -17512.527} C_VEL
LIN {X 0,Y 277.232,Z 303.578,A -85,B 0,C 180,E1 -17516.102,E2 -17516.102} C_VEL
LIN {X 0,Y 277.248,Z 303.555,A -85,B 0,C 180,E1 -17519.537,E2 -17519.537} C_VEL
LIN {X 0,Y 277.341,Z 303.563,A -85,B 0,C 180,E1 -17522.862,E2 -17522.862} C_VEL
LIN {X 0,Y 277.282,Z 303.563,A -85,B 0,C 180,E1 -17526.075,E2 -17526.075} C_VEL
LIN {X 0,Y 277.327,Z 303.561,A -85,B 0,C 180,E1 -17530.765,E2 -17530.765} C_VEL
LIN {X 0,Y 277.413,Z 303.555,A -85,B 0,C 180,E1 -17535.324,E2 -17535.324} C_VEL
LIN {X 0,Y 277.429,Z 303.554,A -85,B 0,C 180,E1 -17538.399,E2 -17538.399} C_VEL
LIN {X 0,Y 278.501,Z 306.466,A -85,B 0,C 180,E1 -17538.692,E2 -17538.692} C_VEL
LIN {X 0,Y 280.278,Z 309.081,A -85,B 0,C 180,E1 -17539.056,E2 -17539.056} C_VEL
LIN {X 0,Y 287.697,Z 320.992,A -85,B 0,C 180,E1 -17540.548,E2 -17540.548} C_VEL
LIN {X 0,Y 291.212,Z 327.598,A -85,B 0,C 180,E1 -17541.257,E2 -17541.257} C_VEL
LIN {X 0,Y 299.977,Z 345.384,A -85,B 0,C 180,E1 -17542.973,E2 -17542.973} C_VEL
LIN {X 0,Y 305.178,Z 357.569,A -85,B 0,C 180,E1 -17543.981,E2 -17543.981} C_VEL
LIN {X 0,Y 300.586,Z 465.015,A -85,B 0,C 180,E1 -17546.607,E2 -17546.607} C_VEL
LIN {X 0,Y 299.336,Z 480.661,A -85,B 0,C 180,E1 -17547.224,E2 -17547.224} C_VEL
LIN {X 0,Y 297.645,Z 496.368,A -85,B 0,C 180,E1 -17548.139,E2 -17548.139} C_VEL
LIN {X 0,Y 295.742,Z 509.984,A -85,B 0,C 180,E1 -17549.19,E2 -17549.19} C_VEL
LIN {X 0,Y 293.544,Z 523.516,A -85,B 0,C 180,E1 -17550.514,E2 -17550.514} C_VEL
LIN {X 0,Y 291.028,Z 536.483,A -85,B 0,C 180,E1 -17552.075,E2 -17552.075} C_VEL
LIN {X 0,Y 288.5,Z 548.415,A -85,B 0,C 180,E1 -17553.835,E2 -17553.835} C_VEL
LIN {X 0,Y 285.736,Z 560.479,A -85,B 0,C 180,E1 -17556,E2 -17556} C_VEL
LIN {X 0,Y 283.475,Z 570.208,A -85,B 0,C 180,E1 -17558.127,E2 -17558.127} C_VEL
LIN {X 0,Y 281.334,Z 579.023,A -85,B 0,C 180,E1 -17560.434,E2 -17560.434} C_VEL
LIN {X 0,Y 279.322,Z 587.368,A -85,B 0,C 180,E1 -17563.087,E2 -17563.087} C_VEL
LIN {X 0,Y 277.712,Z 594.565,A -85,B 0,C 180,E1 -17565.93,E2 -17565.93} C_VEL
LIN {X 0,Y 276.654,Z 599.8,A -85,B 0,C 180,E1 -17568.513,E2 -17568.513} C_VEL
LIN {X 0,Y 276.012,Z 603.591,A -85,B 0,C 180,E1 -17570.883,E2 -17570.883} C_VEL
LIN {X 0,Y 275.449,Z 606.588,A -85,B 0,C 180,E1 -17573.297,E2 -17573.297} C_VEL
LIN {X 0,Y 274.998,Z 609.312,A -85,B 0,C 180,E1 -17576.566,E2 -17576.566} C_VEL
LIN {X 0,Y 274.876,Z 610.555,A -85,B 0,C 180,E1 -17579.629,E2 -17579.629} C_VEL
LIN {X 0,Y 274.954,Z 610.587,A -85,B 0,C 180,E1 -17582.495,E2 -17582.495} C_VEL
LIN {X 0,Y 275.215,Z 609.571,A -85,B 0,C 180,E1 -17585.204,E2 -17585.204} C_VEL
LIN {X 0,Y 275.7,Z 607.722,A -85,B 0,C 180,E1 -17587.798,E2 -17587.798} C_VEL
LIN {X 0,Y 276.47,Z 605.012,A -85,B 0,C 180,E1 -17590.31,E2 -17590.31} C_VEL
LIN {X 0,Y 277.586,Z 600.875,A -85,B 0,C 180,E1 -17593.123,E2 -17593.123} C_VEL
LIN {X 0,Y 279.08,Z 595.631,A -85,B 0,C 180,E1 -17595.866,E2 -17595.866} C_VEL
LIN {X 0,Y 281.081,Z 589.031,A -85,B 0,C 180,E1 -17598.597,E2 -17598.597} C_VEL
LIN {X 0,Y 283.425,Z 581.543,A -85,B 0,C 180,E1 -17601.106,E2 -17601.106} C_VEL
LIN {X 0,Y 286.154,Z 572.687,A -85,B 0,C 180,E1 -17603.539,E2 -17603.539} C_VEL
LIN {X 0,Y 289.129,Z 562.925,A -85,B 0,C 180,E1 -17605.733,E2 -17605.733} C_VEL
LIN {X 0,Y 292.283,Z 551.787,A -85,B 0,C 180,E1 -17607.802,E2 -17607.802} C_VEL
LIN {X 0,Y 295.237,Z 540.529,A -85,B 0,C 180,E1 -17609.523,E2 -17609.523} C_VEL
LIN {X 0,Y 298.083,Z 528.307,A -85,B 0,C 180,E1 -17611.072,E2 -17611.072} C_VEL
LIN {X 0,Y 301.047,Z 514.148,A -85,B 0,C 180,E1 -17612.51,E2 -17612.51} C_VEL
LIN {X 0,Y 303.437,Z 500.104,A -85,B 0,C 180,E1 -17613.64,E2 -17613.64} C_VEL
LIN {X 0,Y 305.489,Z 485.205,A -85,B 0,C 180,E1 -17614.548,E2 -17614.548} C_VEL
LIN {X 0,Y 307.087,Z 469.577,A -85,B 0,C 180,E1 -17615.217,E2 -17615.217} C_VEL
LIN {X 0,Y 308.111,Z 453.014,A -85,B 0,C 180,E1 -17615.677,E2 -17615.677} C_VEL
LIN {X 0,Y 307.883,Z 447.231,A -85,B 0,C 180,E1 -17615.9,E2 -17615.9} C_VEL
LIN {X 0,Y 304.446,Z 428.716,A -85,B 0,C 180,E1 -17617.07,E2 -17617.07} C_VEL
LIN {X 0,Y 304.299,Z 422.933,A -85,B 0,C 180,E1 -17617.289,E2 -17617.289} C_VEL
LIN {X 0,Y 307.379,Z 364.969,A -85,B 0,C 180,E1 -17618.734,E2 -17618.734} C_VEL
LIN {X 0,Y 302.138,Z 353.709,A -85,B 0,C 180,E1 -17620.108,E2 -17620.108} C_VEL
LIN {X 0,Y 294.991,Z 340.317,A -85,B 0,C 180,E1 -17622.076,E2 -17622.076} C_VEL
LIN {X 0,Y 287.226,Z 327.632,A -85,B 0,C 180,E1 -17624.389,E2 -17624.389} C_VEL
LIN {X 0,Y 284.242,Z 323.462,A -85,B 0,C 180,E1 -17625.328,E2 -17625.328} C_VEL
LIN {X 0,Y 281.104,Z 319.184,A -85,B 0,C 180,E1 -17626.365,E2 -17626.365} C_VEL
LIN {X 0,Y 278.48,Z 315.534,A -85,B 0,C 180,E1 -17627.292,E2 -17627.292} C_VEL
LIN {X 0,Y 275.377,Z 312.004,A -85,B 0,C 180,E1 -17628.408,E2 -17628.408} C_VEL
LIN {X 0,Y 274.361,Z 309.962,A -85,B 0,C 180,E1 -17628.833,E2 -17628.833} C_VEL
LIN {X 0,Y 271.902,Z 307.984,A -85,B 0,C 180,E1 -17629.734,E2 -17629.734} C_VEL
LIN {X 0,Y 270.604,Z 305.291,A -85,B 0,C 180,E1 -17630.318,E2 -17630.318} C_VEL
LIN {X 0,Y 270.464,Z 304.422,A -85,B 0,C 180,E1 -17630.45,E2 -17630.45} C_VEL
LIN {X 0,Y 270.588,Z 304.405,A -85,B 0,C 180,E1 -17632.541,E2 -17632.541} C_VEL
LIN {X 0,Y 270.777,Z 304.378,A -85,B 0,C 180,E1 -17638.515,E2 -17638.515} C_VEL
LIN {X 0,Y 270.777,Z 304.375,A -85,B 0,C 180,E1 -17641.49,E2 -17641.49} C_VEL
LIN {X 0,Y 270.562,Z 304.401,A -85,B 0,C 180,E1 -17647.465,E2 -17647.465} C_VEL
LIN {X 0,Y 270.381,Z 304.424,A -85,B 0,C 180,E1 -17650.486,E2 -17650.486} C_VEL
LIN {X 0,Y 270.362,Z 304.43,A -85,B 0,C 180,E1 -17655.069,E2 -17655.069} C_VEL
LIN {X 0,Y 270.218,Z 304.444,A -85,B 0,C 180,E1 -17659.764,E2 -17659.764} C_VEL
LIN {X 0,Y 270.18,Z 304.455,A -85,B 0,C 180,E1 -17664.439,E2 -17664.439} C_VEL
LIN {X 0,Y 270.181,Z 304.452,A -85,B 0,C 180,E1 -17667.921,E2 -17667.921} C_VEL
LIN {X 0,Y 270.166,Z 304.449,A -85,B 0,C 180,E1 -17671.353,E2 -17671.353} C_VEL
LIN {X 0,Y 270.221,Z 304.449,A -85,B 0,C 180,E1 -17675.584,E2 -17675.584} C_VEL
LIN {X 0,Y 270.216,Z 304.448,A -85,B 0,C 180,E1 -17676.269,E2 -17676.269} C_VEL
LIN {X 0,Y 272.678,Z 311.462,A -85,B 0,C 180,E1 -17680.331,E2 -17680.331} C_VEL
LIN {X 0,Y 275.801,Z 316.089,A -85,B 0,C 180,E1 -17681.557,E2 -17681.557} C_VEL
LIN {X 0,Y 277.672,Z 318.618,A -85,B 0,C 180,E1 -17682.248,E2 -17682.248} C_VEL
LIN {X 0,Y 282.117,Z 325.309,A -85,B 0,C 180,E1 -17683.822,E2 -17683.822} C_VEL
LIN {X 0,Y 285.493,Z 330.544,A -85,B 0,C 180,E1 -17684.934,E2 -17684.934} C_VEL
LIN {X 0,Y 288.979,Z 336.348,A -85,B 0,C 180,E1 -17686.034,E2 -17686.034} C_VEL
LIN {X 0,Y 294.301,Z 345.698,A -85,B 0,C 180,E1 -17687.615,E2 -17687.615} C_VEL
LIN {X 0,Y 299.601,Z 356.049,A -85,B 0,C 180,E1 -17689.113,E2 -17689.113} C_VEL
LIN {X 0,Y 306.057,Z 370.584,A -85,B 0,C 180,E1 -17690.852,E2 -17690.852} C_VEL
LIN {X 0,Y 306.972,Z 373.486,A -85,B 0,C 180,E1 -17691.118,E2 -17691.118} C_VEL
LIN {X 0,Y 306.616,Z 382.879,A -85,B 0,C 180,E1 -17691.379,E2 -17691.379} C_VEL
LIN {X 0,Y 301.357,Z 480.294,A -85,B 0,C 180,E1 -17693.822,E2 -17693.822} C_VEL
LIN {X 0,Y 299.605,Z 496.289,A -85,B 0,C 180,E1 -17694.459,E2 -17694.459} C_VEL
LIN {X 0,Y 297.221,Z 511.542,A -85,B 0,C 180,E1 -17695.323,E2 -17695.323} C_VEL
LIN {X 0,Y 294.814,Z 524.872,A -85,B 0,C 180,E1 -17696.342,E2 -17696.342} C_VEL
LIN {X 0,Y 291.761,Z 538.789,A -85,B 0,C 180,E1 -17697.689,E2 -17697.689} C_VEL
LIN {X 0,Y 288.554,Z 551.598,A -85,B 0,C 180,E1 -17699.239,E2 -17699.239} C_VEL
LIN {X 0,Y 284.877,Z 564.952,A -85,B 0,C 180,E1 -17701.246,E2 -17701.246} C_VEL
LIN {X 0,Y 281.524,Z 576.11,A -85,B 0,C 180,E1 -17703.299,E2 -17703.299} C_VEL
LIN {X 0,Y 278.305,Z 586.816,A -85,B 0,C 180,E1 -17705.728,E2 -17705.728} C_VEL
LIN {X 0,Y 275.371,Z 596.048,A -85,B 0,C 180,E1 -17708.281,E2 -17708.281} C_VEL
LIN {X 0,Y 272.735,Z 604.589,A -85,B 0,C 180,E1 -17711.211,E2 -17711.211} C_VEL
LIN {X 0,Y 270.737,Z 611.657,A -85,B 0,C 180,E1 -17714.273,E2 -17714.273} C_VEL
LIN {X 0,Y 269.415,Z 616.935,A -85,B 0,C 180,E1 -17717.19,E2 -17717.19} C_VEL
LIN {X 0,Y 268.733,Z 620.12,A -85,B 0,C 180,E1 -17719.452,E2 -17719.452} C_VEL
LIN {X 0,Y 268.235,Z 623.328,A -85,B 0,C 180,E1 -17722.473,E2 -17722.473} C_VEL
LIN {X 0,Y 268.081,Z 625.328,A -85,B 0,C 180,E1 -17725.49,E2 -17725.49} C_VEL
LIN {X 0,Y 268.185,Z 626.121,A -85,B 0,C 180,E1 -17728.499,E2 -17728.499} C_VEL
LIN {X 0,Y 268.186,Z 625.754,A -85,B 0,C 180,E1 -17731.502,E2 -17731.502} C_VEL
LIN {X 0,Y 268.113,Z 624.207,A -85,B 0,C 180,E1 -17734.511,E2 -17734.511} C_VEL
LIN {X 0,Y 268.25,Z 621.45,A -85,B 0,C 180,E1 -17737.528,E2 -17737.528} C_VEL
LIN {X 0,Y 268.677,Z 617.412,A -85,B 0,C 180,E1 -17740.551,E2 -17740.551} C_VEL
LIN {X 0,Y 269.595,Z 611.975,A -85,B 0,C 180,E1 -17743.569,E2 -17743.569} C_VEL
LIN {X 0,Y 270.967,Z 605.008,A -85,B 0,C 180,E1 -17746.577,E2 -17746.577} C_VEL
LIN {X 0,Y 272.638,Z 597.478,A -85,B 0,C 180,E1 -17749.188,E2 -17749.188} C_VEL
LIN {X 0,Y 274.914,Z 588.435,A -85,B 0,C 180,E1 -17751.758,E2 -17751.758} C_VEL
LIN {X 0,Y 277.297,Z 578.212,A -85,B 0,C 180,E1 -17754.156,E2 -17754.156} C_VEL
LIN {X 0,Y 279.674,Z 568.267,A -85,B 0,C 180,E1 -17756.089,E2 -17756.089} C_VEL
LIN {X 0,Y 282.528,Z 556.365,A -85,B 0,C 180,E1 -17758.003,E2 -17758.003} C_VEL
LIN {X 0,Y 285.25,Z 543.332,A -85,B 0,C 180,E1 -17759.725,E2 -17759.725} C_VEL
LIN {X 0,Y 287.945,Z 529.243,A -85,B 0,C 180,E1 -17761.21,E2 -17761.21} C_VEL
LIN {X 0,Y 290.205,Z 514.971,A -85,B 0,C 180,E1 -17762.399,E2 -17762.399} C_VEL
LIN {X 0,Y 292.224,Z 500.13,A -85,B 0,C 180,E1 -17763.325,E2 -17763.325} C_VEL
LIN {X 0,Y 293.747,Z 484.88,A -85,B 0,C 180,E1 -17764.004,E2 -17764.004} C_VEL
LIN {X 0,Y 294.841,Z 464.502,A -85,B 0,C 180,E1 -17764.583,E2 -17764.583} C_VEL
LIN {X 0,Y 298.839,Z 372.401,A -85,B 0,C 180,E1 -17766.855,E2 -17766.855} C_VEL
LIN {X 0,Y 297.757,Z 365.811,A -85,B 0,C 180,E1 -17767.19,E2 -17767.19} C_VEL
LIN {X 0,Y 289.568,Z 346.74,A -85,B 0,C 180,E1 -17768.868,E2 -17768.868} C_VEL
LIN {X 0,Y 281.396,Z 329.907,A -85,B 0,C 180,E1 -17770.585,E2 -17770.585} C_VEL
LIN {X 0,Y 273.994,Z 316.076,A -85,B 0,C 180,E1 -17772.206,E2 -17772.206} C_VEL
LIN {X 0,Y 272.874,Z 313.708,A -85,B 0,C 180,E1 -17772.488,E2 -17772.488} C_VEL
LIN {X 0,Y 270.136,Z 304.455,A -85,B 0,C 180,E1 -17775.847,E2 -17775.847} C_VEL
LIN {X 0,Y 270.151,Z 304.458,A -85,B 0,C 180,E1 -17779.428,E2 -17779.428} C_VEL
LIN {X 0,Y 270.209,Z 304.459,A -85,B 0,C 180,E1 -17783.255,E2 -17783.255} C_VEL
LIN {X 0,Y 270.203,Z 304.444,A -85,B 0,C 180,E1 -17786.89,E2 -17786.89} C_VEL
LIN {X 0,Y 270.159,Z 304.456,A -85,B 0,C 180,E1 -17790.376,E2 -17790.376} C_VEL
LIN {X 0,Y 270.179,Z 304.454,A -85,B 0,C 180,E1 -17793.753,E2 -17793.753} C_VEL
LIN {X 0,Y 270.182,Z 304.454,A -85,B 0,C 180,E1 -17797.032,E2 -17797.032} C_VEL
LIN {X 0,Y 270.223,Z 304.447,A -85,B 0,C 180,E1 -17800.236,E2 -17800.236} C_VEL
LIN {X 0,Y 270.367,Z 304.417,A -85,B 0,C 180,E1 -17804.931,E2 -17804.931} C_VEL
LIN {X 0,Y 270.385,Z 304.41,A -85,B 0,C 180,E1 -17809.514,E2 -17809.514} C_VEL
LIN {X 0,Y 270.549,Z 304.408,A -85,B 0,C 180,E1 -17812.535,E2 -17812.535} C_VEL
LIN {X 0,Y 270.762,Z 304.357,A -85,B 0,C 180,E1 -17818.51,E2 -17818.51} C_VEL
LIN {X 0,Y 270.765,Z 304.384,A -85,B 0,C 180,E1 -17821.485,E2 -17821.485} C_VEL
LIN {X 0,Y 270.539,Z 304.369,A -85,B 0,C 180,E1 -17827.461,E2 -17827.461} C_VEL
LIN {X 0,Y 270.402,Z 304.424,A -85,B 0,C 180,E1 -17830.48,E2 -17830.48} C_VEL
LIN {X 0,Y 270.361,Z 304.404,A -85,B 0,C 180,E1 -17835.064,E2 -17835.064} C_VEL
LIN {X 0,Y 270.249,Z 304.431,A -85,B 0,C 180,E1 -17839.757,E2 -17839.757} C_VEL
LIN {X 0,Y 270.17,Z 304.44,A -85,B 0,C 180,E1 -17844.592,E2 -17844.592} C_VEL
LIN {X 0,Y 270.175,Z 304.418,A -85,B 0,C 180,E1 -17847.916,E2 -17847.916} C_VEL
LIN {X 0,Y 270.159,Z 304.457,A -85,B 0,C 180,E1 -17851.348,E2 -17851.348} C_VEL
LIN {X 0,Y 270.186,Z 304.432,A -85,B 0,C 180,E1 -17854.904,E2 -17854.904} C_VEL
LIN {X 0,Y 270.187,Z 304.438,A -85,B 0,C 180,E1 -17858.708,E2 -17858.708} C_VEL
LIN {X 0,Y 270.135,Z 304.45,A -85,B 0,C 180,E1 -17863.243,E2 -17863.243} C_VEL
LIN {X 0,Y 270.159,Z 304.447,A -85,B 0,C 180,E1 -17867.44,E2 -17867.44} C_VEL
LIN {X 0,Y 270.194,Z 304.444,A -85,B 0,C 180,E1 -17871.372,E2 -17871.372} C_VEL
LIN {X 0,Y 270.185,Z 304.449,A -85,B 0,C 180,E1 -17875.092,E2 -17875.092} C_VEL
LIN {X 0,Y 270.17,Z 304.437,A -85,B 0,C 180,E1 -17879.135,E2 -17879.135} C_VEL
LIN {X 0,Y 270.249,Z 304.446,A -85,B 0,C 180,E1 -17882.145,E2 -17882.145} C_VEL
LIN {X 0,Y 270.222,Z 304.438,A -85,B 0,C 180,E1 -17885.537,E2 -17885.537} C_VEL
LIN {X 0,Y 270.285,Z 304.434,A -85,B 0,C 180,E1 -17890.243,E2 -17890.243} C_VEL
LIN {X 0,Y 270.381,Z 304.431,A -85,B 0,C 180,E1 -17894.934,E2 -17894.934} C_VEL
LIN {X 0,Y 270.353,Z 304.428,A -85,B 0,C 180,E1 -17897.267,E2 -17897.267} C_VEL
LIN {X 0,Y 271.396,Z 307.347,A -85,B 0,C 180,E1 -17897.576,E2 -17897.576} C_VEL
LIN {X 0,Y 273.081,Z 309.566,A -85,B 0,C 180,E1 -17897.933,E2 -17897.933} C_VEL
LIN {X 0,Y 283.922,Z 327.152,A -85,B 0,C 180,E1 -17900.205,E2 -17900.205} C_VEL
LIN {X 0,Y 294.626,Z 348.945,A -85,B 0,C 180,E1 -17902.388,E2 -17902.388} C_VEL
LIN {X 0,Y 299.137,Z 359.463,A -85,B 0,C 180,E1 -17903.293,E2 -17903.293} C_VEL
LIN {X 0,Y 294.433,Z 465.608,A -85,B 0,C 180,E1 -17905.936,E2 -17905.936} C_VEL
LIN {X 0,Y 293.149,Z 481.086,A -85,B 0,C 180,E1 -17906.563,E2 -17906.563} C_VEL
LIN {X 0,Y 291.549,Z 495.474,A -85,B 0,C 180,E1 -17907.409,E2 -17907.409} C_VEL
LIN {X 0,Y 289.625,Z 508.83,A -85,B 0,C 180,E1 -17908.435,E2 -17908.435} C_VEL
LIN {X 0,Y 287.345,Z 522.589,A -85,B 0,C 180,E1 -17909.777,E2 -17909.777} C_VEL
LIN {X 0,Y 284.956,Z 534.758,A -85,B 0,C 180,E1 -17911.236,E2 -17911.236} C_VEL
LIN {X 0,Y 282.224,Z 547.408,A -85,B 0,C 180,E1 -17913.09,E2 -17913.09} C_VEL
LIN {X 0,Y 279.631,Z 558.404,A -85,B 0,C 180,E1 -17915.046,E2 -17915.046} C_VEL
LIN {X 0,Y 277.152,Z 568.798,A -85,B 0,C 180,E1 -17917.283,E2 -17917.283} C_VEL
LIN {X 0,Y 274.926,Z 577.643,A -85,B 0,C 180,E1 -17919.564,E2 -17919.564} C_VEL
LIN {X 0,Y 272.974,Z 585.382,A -85,B 0,C 180,E1 -17921.961,E2 -17921.961} C_VEL
LIN {X 0,Y 271.479,Z 591.469,A -85,B 0,C 180,E1 -17924.236,E2 -17924.236} C_VEL
LIN {X 0,Y 270.317,Z 596.831,A -85,B 0,C 180,E1 -17926.617,E2 -17926.617} C_VEL
LIN {X 0,Y 269.151,Z 602.52,A -85,B 0,C 180,E1 -17929.842,E2 -17929.842} C_VEL
LIN {X 0,Y 268.776,Z 604.79,A -85,B 0,C 180,E1 -17931.473,E2 -17931.473} C_VEL
LIN {X 0,Y 268.095,Z 608.273,A -85,B 0,C 180,E1 -17934.798,E2 -17934.798} C_VEL
LIN {X 0,Y 267.864,Z 609.687,A -85,B 0,C 180,E1 -17936.874,E2 -17936.874} C_VEL
LIN {X 0,Y 267.779,Z 610.796,A -85,B 0,C 180,E1 -17939.998,E2 -17939.998} C_VEL
LIN {X 0,Y 267.923,Z 610.587,A -85,B 0,C 180,E1 -17943.424,E2 -17943.424} C_VEL
LIN {X 0,Y 268.218,Z 609.648,A -85,B 0,C 180,E1 -17945.687,E2 -17945.687} C_VEL
LIN {X 0,Y 268.886,Z 607.217,A -85,B 0,C 180,E1 -17948.849,E2 -17948.849} C_VEL
LIN {X 0,Y 269.829,Z 603.935,A -85,B 0,C 180,E1 -17951.66,E2 -17951.66} C_VEL
LIN {X 0,Y 271.15,Z 599.648,A -85,B 0,C 180,E1 -17954.41,E2 -17954.41} C_VEL
LIN {X 0,Y 272.86,Z 594.071,A -85,B 0,C 180,E1 -17957.195,E2 -17957.195} C_VEL
LIN {X 0,Y 275.182,Z 586.952,A -85,B 0,C 180,E1 -17960.01,E2 -17960.01} C_VEL
LIN {X 0,Y 277.878,Z 578.729,A -85,B 0,C 180,E1 -17962.631,E2 -17962.631} C_VEL
LIN {X 0,Y 280.946,Z 569.274,A -85,B 0,C 180,E1 -17965.086,E2 -17965.086} C_VEL
LIN {X 0,Y 284.432,Z 557.976,A -85,B 0,C 180,E1 -17967.476,E2 -17967.476} C_VEL
LIN {X 0,Y 288.052,Z 545.381,A -85,B 0,C 180,E1 -17969.627,E2 -17969.627} C_VEL
LIN {X 0,Y 291.564,Z 531.722,A -85,B 0,C 180,E1 -17971.497,E2 -17971.497} C_VEL
LIN {X 0,Y 294.465,Z 518.918,A -85,B 0,C 180,E1 -17972.908,E2 -17972.908} C_VEL
LIN {X 0,Y 297.318,Z 503.763,A -85,B 0,C 180,E1 -17974.227,E2 -17974.227} C_VEL
LIN {X 0,Y 299.567,Z 488.807,A -85,B 0,C 180,E1 -17975.215,E2 -17975.215} C_VEL
LIN {X 0,Y 301.312,Z 473.522,A -85,B 0,C 180,E1 -17975.939,E2 -17975.939} C_VEL
LIN {X 0,Y 302.458,Z 457.329,A -85,B 0,C 180,E1 -17976.443,E2 -17976.443} C_VEL
LIN {X 0,Y 304.299,Z 422.933,A -85,B 0,C 180,E1 -17977.289,E2 -17977.289} C_VEL
LIN {X 0,Y 304.147,Z 417.146,A -85,B 0,C 180,E1 -17977.512,E2 -17977.512} C_VEL
LIN {X 0,Y 300.855,Z 398.659,A -85,B 0,C 180,E1 -17978.74,E2 -17978.74} C_VEL
LIN {X 0,Y 300.716,Z 392.874,A -85,B 0,C 180,E1 -17978.971,E2 -17978.971} C_VEL
LIN {X 0,Y 302.163,Z 367.423,A -85,B 0,C 180,E1 -17979.61,E2 -17979.61} C_VEL
LIN {X 0,Y 296.35,Z 355.005,A -85,B 0,C 180,E1 -17981.22,E2 -17981.22} C_VEL
LIN {X 0,Y 289.271,Z 342.075,A -85,B 0,C 180,E1 -17983.288,E2 -17983.288} C_VEL
LIN {X 0,Y 283.621,Z 332.783,A -85,B 0,C 180,E1 -17985.074,E2 -17985.074} C_VEL
LIN {X 0,Y 278.048,Z 324.937,A -85,B 0,C 180,E1 -17986.958,E2 -17986.958} C_VEL
LIN {X 0,Y 274.88,Z 320.7,A -85,B 0,C 180,E1 -17988.118,E2 -17988.118} C_VEL
LIN {X 0,Y 272.275,Z 317.399,A -85,B 0,C 180,E1 -17989.111,E2 -17989.111} C_VEL
LIN {X 0,Y 271.176,Z 315.879,A -85,B 0,C 180,E1 -17989.55,E2 -17989.55} C_VEL
LIN {X 0,Y 268.844,Z 313.402,A -85,B 0,C 180,E1 -17990.482,E2 -17990.482} C_VEL
LIN {X 0,Y 267.603,Z 310.873,A -85,B 0,C 180,E1 -17991.082,E2 -17991.082} C_VEL
LIN {X 0,Y 265.118,Z 308.97,A -85,B 0,C 180,E1 -17992.147,E2 -17992.147} C_VEL
LIN {X 0,Y 263.794,Z 306.513,A -85,B 0,C 180,E1 -17992.829,E2 -17992.829} C_VEL
LIN {X 0,Y 263.517,Z 305.284,A -85,B 0,C 180,E1 -17993.062,E2 -17993.062} C_VEL
LIN {X 0,Y 263.742,Z 305.254,A -85,B 0,C 180,E1 -17998.476,E2 -17998.476} C_VEL
LIN {X 0,Y 263.741,Z 305.252,A -85,B 0,C 180,E1 -18001.529,E2 -18001.529} C_VEL
LIN {X 0,Y 263.525,Z 305.277,A -85,B 0,C 180,E1 -18007.665,E2 -18007.665} C_VEL
LIN {X 0,Y 263.327,Z 305.302,A -85,B 0,C 180,E1 -18010.77,E2 -18010.77} C_VEL
LIN {X 0,Y 263.304,Z 305.313,A -85,B 0,C 180,E1 -18015.483,E2 -18015.483} C_VEL
LIN {X 0,Y 263.204,Z 305.317,A -85,B 0,C 180,E1 -18020.314,E2 -18020.314} C_VEL
LIN {X 0,Y 263.118,Z 305.33,A -85,B 0,C 180,E1 -18025.303,E2 -18025.303} C_VEL
LIN {X 0,Y 263.114,Z 305.327,A -85,B 0,C 180,E1 -18028.74,E2 -18028.74} C_VEL
LIN {X 0,Y 263.162,Z 305.327,A -85,B 0,C 180,E1 -18033.196,E2 -18033.196} C_VEL
LIN {X 0,Y 263.186,Z 305.474,A -85,B 0,C 180,E1 -18033.98,E2 -18033.98} C_VEL
LIN {X 0,Y 265.263,Z 311.094,A -85,B 0,C 180,E1 -18037.666,E2 -18037.666} C_VEL
LIN {X 0,Y 268.838,Z 316.203,A -85,B 0,C 180,E1 -18039.301,E2 -18039.301} C_VEL
LIN {X 0,Y 270.194,Z 317.998,A -85,B 0,C 180,E1 -18039.862,E2 -18039.862} C_VEL
LIN {X 0,Y 275.071,Z 324.996,A -85,B 0,C 180,E1 -18041.784,E2 -18041.784} C_VEL
LIN {X 0,Y 278.989,Z 331.016,A -85,B 0,C 180,E1 -18043.228,E2 -18043.228} C_VEL
LIN {X 0,Y 282.304,Z 336.248,A -85,B 0,C 180,E1 -18044.366,E2 -18044.366} C_VEL
LIN {X 0,Y 287.259,Z 344.702,A -85,B 0,C 180,E1 -18045.975,E2 -18045.975} C_VEL
LIN {X 0,Y 294.074,Z 357.615,A -85,B 0,C 180,E1 -18048.03,E2 -18048.03} C_VEL
LIN {X 0,Y 300.156,Z 371.378,A -85,B 0,C 180,E1 -18049.78,E2 -18049.78} C_VEL
LIN {X 0,Y 301.866,Z 375.451,A -85,B 0,C 180,E1 -18050.251,E2 -18050.251} C_VEL
LIN {X 0,Y 296.052,Z 479.519,A -85,B 0,C 180,E1 -18052.908,E2 -18052.908} C_VEL
LIN {X 0,Y 294.37,Z 494.896,A -85,B 0,C 180,E1 -18053.515,E2 -18053.515} C_VEL
LIN {X 0,Y 291.897,Z 510.45,A -85,B 0,C 180,E1 -18054.385,E2 -18054.385} C_VEL
LIN {X 0,Y 289.348,Z 523.922,A -85,B 0,C 180,E1 -18055.408,E2 -18055.408} C_VEL
LIN {X 0,Y 286.071,Z 538.5,A -85,B 0,C 180,E1 -18056.828,E2 -18056.828} C_VEL
LIN {X 0,Y 282.497,Z 552.125,A -85,B 0,C 180,E1 -18058.505,E2 -18058.505} C_VEL
LIN {X 0,Y 278.991,Z 564.336,A -85,B 0,C 180,E1 -18060.373,E2 -18060.373} C_VEL
LIN {X 0,Y 275.171,Z 576.356,A -85,B 0,C 180,E1 -18062.632,E2 -18062.632} C_VEL
LIN {X 0,Y 271.725,Z 587.208,A -85,B 0,C 180,E1 -18065.174,E2 -18065.174} C_VEL
LIN {X 0,Y 268.756,Z 596.144,A -85,B 0,C 180,E1 -18067.719,E2 -18067.719} C_VEL
LIN {X 0,Y 265.985,Z 604.622,A -85,B 0,C 180,E1 -18070.715,E2 -18070.715} C_VEL
LIN {X 0,Y 263.919,Z 611.303,A -85,B 0,C 180,E1 -18073.674,E2 -18073.674} C_VEL
LIN {X 0,Y 262.456,Z 616.875,A -85,B 0,C 180,E1 -18076.844,E2 -18076.844} C_VEL
LIN {X 0,Y 261.699,Z 620.019,A -85,B 0,C 180,E1 -18079.166,E2 -18079.166} C_VEL
LIN {X 0,Y 261.151,Z 623.188,A -85,B 0,C 180,E1 -18082.268,E2 -18082.268} C_VEL
LIN {X 0,Y 260.984,Z 625.164,A -85,B 0,C 180,E1 -18085.367,E2 -18085.367} C_VEL
LIN {X 0,Y 261.111,Z 625.927,A -85,B 0,C 180,E1 -18088.458,E2 -18088.458} C_VEL
LIN {X 0,Y 261.113,Z 625.52,A -85,B 0,C 180,E1 -18091.543,E2 -18091.543} C_VEL
LIN {X 0,Y 261.024,Z 623.932,A -85,B 0,C 180,E1 -18094.634,E2 -18094.634} C_VEL
LIN {X 0,Y 261.182,Z 621.132,A -85,B 0,C 180,E1 -18097.733,E2 -18097.733} C_VEL
LIN {X 0,Y 261.642,Z 617.048,A -85,B 0,C 180,E1 -18100.838,E2 -18100.838} C_VEL
LIN {X 0,Y 262.603,Z 611.57,A -85,B 0,C 180,E1 -18103.938,E2 -18103.938} C_VEL
LIN {X 0,Y 264.077,Z 604.547,A -85,B 0,C 180,E1 -18107.023,E2 -18107.023} C_VEL
LIN {X 0,Y 265.844,Z 596.976,A -85,B 0,C 180,E1 -18109.698,E2 -18109.698} C_VEL
LIN {X 0,Y 268.272,Z 587.871,A -85,B 0,C 180,E1 -18112.325,E2 -18112.325} C_VEL
LIN {X 0,Y 270.9,Z 577.052,A -85,B 0,C 180,E1 -18114.893,E2 -18114.893} C_VEL
LIN {X 0,Y 273.741,Z 565.556,A -85,B 0,C 180,E1 -18117.111,E2 -18117.111} C_VEL
LIN {X 0,Y 276.685,Z 553.138,A -85,B 0,C 180,E1 -18119.064,E2 -18119.064} C_VEL
LIN {X 0,Y 279.601,Z 539.452,A -85,B 0,C 180,E1 -18120.807,E2 -18120.807} C_VEL
LIN {X 0,Y 282.306,Z 525.375,A -85,B 0,C 180,E1 -18122.224,E2 -18122.224} C_VEL
LIN {X 0,Y 284.558,Z 511.308,A -85,B 0,C 180,E1 -18123.335,E2 -18123.335} C_VEL
LIN {X 0,Y 286.545,Z 496.031,A -85,B 0,C 180,E1 -18124.234,E2 -18124.234} C_VEL
LIN {X 0,Y 288.016,Z 479.931,A -85,B 0,C 180,E1 -18124.883,E2 -18124.883} C_VEL
LIN {X 0,Y 292.856,Z 373.265,A -85,B 0,C 180,E1 -18127.592,E2 -18127.592} C_VEL
LIN {X 0,Y 291.967,Z 368.232,A -85,B 0,C 180,E1 -18127.867,E2 -18127.867} C_VEL
LIN {X 0,Y 283.838,Z 349.382,A -85,B 0,C 180,E1 -18129.583,E2 -18129.583} C_VEL
LIN {X 0,Y 275.978,Z 333.099,A -85,B 0,C 180,E1 -18131.3,E2 -18131.3} C_VEL
LIN {X 0,Y 267.399,Z 317.115,A -85,B 0,C 180,E1 -18133.254,E2 -18133.254} C_VEL
LIN {X 0,Y 265.509,Z 313.361,A -85,B 0,C 180,E1 -18133.764,E2 -18133.764} C_VEL
LIN {X 0,Y 263.116,Z 305.327,A -85,B 0,C 180,E1 -18136.825,E2 -18136.825} C_VEL
LIN {X 0,Y 263.116,Z 305.326,A -85,B 0,C 180,E1 -18140.769,E2 -18140.769} C_VEL
LIN {X 0,Y 263.158,Z 305.325,A -85,B 0,C 180,E1 -18144.015,E2 -18144.015} C_VEL
LIN {X 0,Y 263.128,Z 305.332,A -85,B 0,C 180,E1 -18147.709,E2 -18147.709} C_VEL
LIN {X 0,Y 263.138,Z 305.332,A -85,B 0,C 180,E1 -18151.808,E2 -18151.808} C_VEL
LIN {X 0,Y 263.115,Z 305.333,A -85,B 0,C 180,E1 -18156.378,E2 -18156.378} C_VEL
LIN {X 0,Y 263.209,Z 305.324,A -85,B 0,C 180,E1 -18159.687,E2 -18159.687} C_VEL
LIN {X 0,Y 263.31,Z 305.303,A -85,B 0,C 180,E1 -18164.517,E2 -18164.517} C_VEL
LIN {X 0,Y 263.331,Z 305.284,A -85,B 0,C 180,E1 -18169.23,E2 -18169.23} C_VEL
LIN {X 0,Y 263.511,Z 305.285,A -85,B 0,C 180,E1 -18172.334,E2 -18172.334} C_VEL
LIN {X 0,Y 263.724,Z 305.232,A -85,B 0,C 180,E1 -18178.47,E2 -18178.47} C_VEL
LIN {X 0,Y 263.729,Z 305.26,A -85,B 0,C 180,E1 -18181.524,E2 -18181.524} C_VEL
LIN {X 0,Y 263.502,Z 305.247,A -85,B 0,C 180,E1 -18187.661,E2 -18187.661} C_VEL
LIN {X 0,Y 263.342,Z 305.304,A -85,B 0,C 180,E1 -18190.764,E2 -18190.764} C_VEL
LIN {X 0,Y 263.304,Z 305.278,A -85,B 0,C 180,E1 -18195.478,E2 -18195.478} C_VEL
LIN {X 0,Y 263.229,Z 305.314,A -85,B 0,C 180,E1 -18200.306,E2 -18200.306} C_VEL
LIN {X 0,Y 263.112,Z 305.309,A -85,B 0,C 180,E1 -18205.298,E2 -18205.298} C_VEL
LIN {X 0,Y 263.108,Z 305.307,A -85,B 0,C 180,E1 -18208.735,E2 -18208.735} C_VEL
LIN {X 0,Y 263.116,Z 305.334,A -85,B 0,C 180,E1 -18212.287,E2 -18212.287} C_VEL
LIN {X 0,Y 263.144,Z 305.297,A -85,B 0,C 180,E1 -18215.981,E2 -18215.981} C_VEL
LIN {X 0,Y 263.08,Z 305.337,A -85,B 0,C 180,E1 -18219.873,E2 -18219.873} C_VEL
LIN {X 0,Y 263.07,Z 305.32,A -85,B 0,C 180,E1 -18223.991,E2 -18223.991} C_VEL
LIN {X 0,Y 263.112,Z 305.335,A -85,B 0,C 180,E1 -18228.405,E2 -18228.405} C_VEL
LIN {X 0,Y 263.144,Z 305.313,A -85,B 0,C 180,E1 -18232.101,E2 -18232.101} C_VEL
LIN {X 0,Y 263.138,Z 305.334,A -85,B 0,C 180,E1 -18235.884,E2 -18235.884} C_VEL
LIN {X 0,Y 263.115,Z 305.314,A -85,B 0,C 180,E1 -18239.502,E2 -18239.502} C_VEL
LIN {X 0,Y 263.176,Z 305.326,A -85,B 0,C 180,E1 -18243.001,E2 -18243.001} C_VEL
LIN {X 0,Y 263.14,Z 305.328,A -85,B 0,C 180,E1 -18246.383,E2 -18246.383} C_VEL
LIN {X 0,Y 263.248,Z 305.308,A -85,B 0,C 180,E1 -18249.692,E2 -18249.692} C_VEL
LIN {X 0,Y 263.329,Z 305.304,A -85,B 0,C 180,E1 -18254.52,E2 -18254.52} C_VEL
LIN {X 0,Y 263.303,Z 305.306,A -85,B 0,C 180,E1 -18256.1,E2 -18256.1} C_VEL
LIN {X 0,Y 264.399,Z 308.306,A -85,B 0,C 180,E1 -18256.419,E2 -18256.419} C_VEL
LIN {X 0,Y 266.155,Z 310.681,A -85,B 0,C 180,E1 -18256.81,E2 -18256.81} C_VEL
LIN {X 0,Y 277.347,Z 328.6,A -85,B 0,C 180,E1 -18259.269,E2 -18259.269} C_VEL
LIN {X 0,Y 280.835,Z 335.08,A -85,B 0,C 180,E1 -18260.014,E2 -18260.014} C_VEL
LIN {X 0,Y 289.534,Z 353.017,A -85,B 0,C 180,E1 -18261.832,E2 -18261.832} C_VEL
LIN {X 0,Y 293.068,Z 361.269,A -85,B 0,C 180,E1 -18262.564,E2 -18262.564} C_VEL
LIN {X 0,Y 290.523,Z 418.727,A -85,B 0,C 180,E1 -18264.011,E2 -18264.011} C_VEL
LIN {X 0,Y 288.307,Z 466.191,A -85,B 0,C 180,E1 -18265.236,E2 -18265.236} C_VEL
LIN {X 0,Y 286.907,Z 482.306,A -85,B 0,C 180,E1 -18265.917,E2 -18265.917} C_VEL
LIN {X 0,Y 285.181,Z 497.078,A -85,B 0,C 180,E1 -18266.821,E2 -18266.821} C_VEL
LIN {X 0,Y 283.209,Z 510.177,A -85,B 0,C 180,E1 -18267.866,E2 -18267.866} C_VEL
LIN {X 0,Y 280.857,Z 523.797,A -85,B 0,C 180,E1 -18269.245,E2 -18269.245} C_VEL
LIN {X 0,Y 278.095,Z 537.079,A -85,B 0,C 180,E1 -18270.904,E2 -18270.904} C_VEL
LIN {X 0,Y 275.391,Z 549.009,A -85,B 0,C 180,E1 -18272.742,E2 -18272.742} C_VEL
LIN {X 0,Y 272.653,Z 560.084,A -85,B 0,C 180,E1 -18274.805,E2 -18274.805} C_VEL
LIN {X 0,Y 270.14,Z 570.233,A -85,B 0,C 180,E1 -18277.098,E2 -18277.098} C_VEL
LIN {X 0,Y 267.506,Z 580.19,A -85,B 0,C 180,E1 -18279.832,E2 -18279.832} C_VEL
LIN {X 0,Y 265.37,Z 588.408,A -85,B 0,C 180,E1 -18282.62,E2 -18282.62} C_VEL
LIN {X 0,Y 263.705,Z 595.159,A -85,B 0,C 180,E1 -18285.456,E2 -18285.456} C_VEL
LIN {X 0,Y 262.382,Z 601.29,A -85,B 0,C 180,E1 -18288.748,E2 -18288.748} C_VEL
LIN {X 0,Y 261.722,Z 604.893,A -85,B 0,C 180,E1 -18291.254,E2 -18291.254} C_VEL
LIN {X 0,Y 261.172,Z 607.66,A -85,B 0,C 180,E1 -18293.814,E2 -18293.814} C_VEL
LIN {X 0,Y 260.727,Z 610.101,A -85,B 0,C 180,E1 -18297.272,E2 -18297.272} C_VEL
LIN {X 0,Y 260.679,Z 611.037,A -85,B 0,C 180,E1 -18300.382,E2 -18300.382} C_VEL
LIN {X 0,Y 260.838,Z 610.866,A -85,B 0,C 180,E1 -18303.363,E2 -18303.363} C_VEL
LIN {X 0,Y 261.208,Z 609.679,A -85,B 0,C 180,E1 -18306.292,E2 -18306.292} C_VEL
LIN {X 0,Y 261.794,Z 607.704,A -85,B 0,C 180,E1 -18308.88,E2 -18308.88} C_VEL
LIN {X 0,Y 262.853,Z 604.319,A -85,B 0,C 180,E1 -18311.944,E2 -18311.944} C_VEL
LIN {X 0,Y 264.286,Z 599.988,A -85,B 0,C 180,E1 -18314.827,E2 -18314.827} C_VEL
LIN {X 0,Y 266.12,Z 594.421,A -85,B 0,C 180,E1 -18317.683,E2 -18317.683} C_VEL
LIN {X 0,Y 268.802,Z 586.693,A -85,B 0,C 180,E1 -18320.803,E2 -18320.803} C_VEL
LIN {X 0,Y 271.658,Z 578.334,A -85,B 0,C 180,E1 -18323.489,E2 -18323.489} C_VEL
LIN {X 0,Y 274.848,Z 569.055,A -85,B 0,C 180,E1 -18325.915,E2 -18325.915} C_VEL
LIN {X 0,Y 278.354,Z 558.236,A -85,B 0,C 180,E1 -18328.237,E2 -18328.237} C_VEL
LIN {X 0,Y 281.713,Z 547.079,A -85,B 0,C 180,E1 -18330.195,E2 -18330.195} C_VEL
LIN {X 0,Y 284.887,Z 535.482,A -85,B 0,C 180,E1 -18331.873,E2 -18331.873} C_VEL
LIN {X 0,Y 287.948,Z 522.904,A -85,B 0,C 180,E1 -18333.365,E2 -18333.365} C_VEL
LIN {X 0,Y 291.006,Z 508.269,A -85,B 0,C 180,E1 -18334.744,E2 -18334.744} C_VEL
LIN {X 0,Y 293.31,Z 494.518,A -85,B 0,C 180,E1 -18335.758,E2 -18335.758} C_VEL
LIN {X 0,Y 295.37,Z 479.241,A -85,B 0,C 180,E1 -18336.589,E2 -18336.589} C_VEL
LIN {X 0,Y 296.779,Z 464.029,A -85,B 0,C 180,E1 -18337.154,E2 -18337.154} C_VEL
LIN {X 0,Y 300.716,Z 392.874,A -85,B 0,C 180,E1 -18338.971,E2 -18338.971} C_VEL
LIN {X 0,Y 300.704,Z 387.033,A -85,B 0,C 180,E1 -18339.182,E2 -18339.182} C_VEL
LIN {X 0,Y 299.658,Z 379.549,A -85,B 0,C 180,E1 -18339.649,E2 -18339.649} C_VEL
LIN {X 0,Y 298.279,Z 374.215,A -85,B 0,C 180,E1 -18340.111,E2 -18340.111} C_VEL
LIN {X 0,Y 297.149,Z 370.807,A -85,B 0,C 180,E1 -18340.461,E2 -18340.461} C_VEL
LIN {X 0,Y 294.513,Z 364.363,A -85,B 0,C 180,E1 -18341.246,E2 -18341.246} C_VEL
LIN {X 0,Y 289.06,Z 353.479,A -85,B 0,C 180,E1 -18342.867,E2 -18342.867} C_VEL
LIN {X 0,Y 283.081,Z 342.828,A -85,B 0,C 180,E1 -18344.769,E2 -18344.769} C_VEL
LIN {X 0,Y 279.474,Z 337.012,A -85,B 0,C 180,E1 -18345.983,E2 -18345.983} C_VEL
LIN {X 0,Y 274.67,Z 330.247,A -85,B 0,C 180,E1 -18347.699,E2 -18347.699} C_VEL
LIN {X 0,Y 271.956,Z 326.555,A -85,B 0,C 180,E1 -18348.733,E2 -18348.733} C_VEL
LIN {X 0,Y 269.145,Z 322.738,A -85,B 0,C 180,E1 -18349.86,E2 -18349.86} C_VEL
LIN {X 0,Y 265.979,Z 318.93,A -85,B 0,C 180,E1 -18351.212,E2 -18351.212} C_VEL
LIN {X 0,Y 264.845,Z 317.067,A -85,B 0,C 180,E1 -18351.757,E2 -18351.757} C_VEL
LIN {X 0,Y 262.389,Z 314.656,A -85,B 0,C 180,E1 -18352.884,E2 -18352.884} C_VEL
LIN {X 0,Y 260.994,Z 311.926,A -85,B 0,C 180,E1 -18353.642,E2 -18353.642} C_VEL
LIN {X 0,Y 258.166,Z 310.116,A -85,B 0,C 180,E1 -18355.025,E2 -18355.025} C_VEL
LIN {X 0,Y 256.847,Z 307.962,A -85,B 0,C 180,E1 -18355.835,E2 -18355.835} C_VEL
LIN {X 0,Y 256.423,Z 306.164,A -85,B 0,C 180,E1 -18356.27,E2 -18356.27} C_VEL
LIN {X 0,Y 256.705,Z 306.131,A -85,B 0,C 180,E1 -18358.434,E2 -18358.434} C_VEL
LIN {X 0,Y 256.704,Z 306.128,A -85,B 0,C 180,E1 -18361.571,E2 -18361.571} C_VEL
LIN {X 0,Y 256.455,Z 306.166,A -85,B 0,C 180,E1 -18366.296,E2 -18366.296} C_VEL
LIN {X 0,Y 256.396,Z 306.174,A -85,B 0,C 180,E1 -18369.469,E2 -18369.469} C_VEL
LIN {X 0,Y 256.225,Z 306.186,A -85,B 0,C 180,E1 -18374.294,E2 -18374.294} C_VEL
LIN {X 0,Y 256.157,Z 306.195,A -85,B 0,C 180,E1 -18377.568,E2 -18377.568} C_VEL
LIN {X 0,Y 256.115,Z 306.204,A -85,B 0,C 180,E1 -18381.1,E2 -18381.1} C_VEL
LIN {X 0,Y 256.08,Z 306.209,A -85,B 0,C 180,E1 -18385.09,E2 -18385.09} C_VEL
LIN {X 0,Y 256.073,Z 306.204,A -85,B 0,C 180,E1 -18388.572,E2 -18388.572} C_VEL
LIN {X 0,Y 256.104,Z 306.3,A -85,B 0,C 180,E1 -18391.084,E2 -18391.084} C_VEL
LIN {X 0,Y 257.736,Z 310.552,A -85,B 0,C 180,E1 -18394.428,E2 -18394.428} C_VEL
LIN {X 0,Y 262.023,Z 316.326,A -85,B 0,C 180,E1 -18396.697,E2 -18396.697} C_VEL
LIN {X 0,Y 263.703,Z 318.655,A -85,B 0,C 180,E1 -18397.52,E2 -18397.52} C_VEL
LIN {X 0,Y 267.446,Z 323.915,A -85,B 0,C 180,E1 -18399.243,E2 -18399.243} C_VEL
LIN {X 0,Y 272.233,Z 330.896,A -85,B 0,C 180,E1 -18401.206,E2 -18401.206} C_VEL
LIN {X 0,Y 278.053,Z 340.037,A -85,B 0,C 180,E1 -18403.392,E2 -18403.392} C_VEL
LIN {X 0,Y 284.047,Z 350.604,A -85,B 0,C 180,E1 -18405.441,E2 -18405.441} C_VEL
LIN {X 0,Y 290.356,Z 362.985,A -85,B 0,C 180,E1 -18407.434,E2 -18407.434} C_VEL
LIN {X 0,Y 295.816,Z 375.721,A -85,B 0,C 180,E1 -18409.087,E2 -18409.087} C_VEL
LIN {X 0,Y 296.738,Z 377.875,A -85,B 0,C 180,E1 -18409.352,E2 -18409.352} C_VEL
LIN {X 0,Y 290.834,Z 479.082,A -85,B 0,C 180,E1 -18411.962,E2 -18411.962} C_VEL
LIN {X 0,Y 288.988,Z 495.27,A -85,B 0,C 180,E1 -18412.613,E2 -18412.613} C_VEL
LIN {X 0,Y 286.444,Z 510.618,A -85,B 0,C 180,E1 -18413.49,E2 -18413.49} C_VEL
LIN {X 0,Y 284.012,Z 523.025,A -85,B 0,C 180,E1 -18414.444,E2 -18414.444} C_VEL
LIN {X 0,Y 280.767,Z 536.845,A -85,B 0,C 180,E1 -18415.78,E2 -18415.78} C_VEL
LIN {X 0,Y 277.576,Z 548.883,A -85,B 0,C 180,E1 -18417.236,E2 -18417.236} C_VEL
LIN {X 0,Y 273.858,Z 561.59,A -85,B 0,C 180,E1 -18419.12,E2 -18419.12} C_VEL
LIN {X 0,Y 270.059,Z 573.178,A -85,B 0,C 180,E1 -18421.222,E2 -18421.222} C_VEL
LIN {X 0,Y 266.444,Z 584.005,A -85,B 0,C 180,E1 -18423.655,E2 -18423.655} C_VEL
LIN {X 0,Y 263.093,Z 593.832,A -85,B 0,C 180,E1 -18426.38,E2 -18426.38} C_VEL
LIN {X 0,Y 260.236,Z 601.682,A -85,B 0,C 180,E1 -18429.034,E2 -18429.034} C_VEL
LIN {X 0,Y 258.011,Z 608.244,A -85,B 0,C 180,E1 -18431.746,E2 -18431.746} C_VEL
LIN {X 0,Y 256.157,Z 614.306,A -85,B 0,C 180,E1 -18434.893,E2 -18434.893} C_VEL
LIN {X 0,Y 254.867,Z 619.002,A -85,B 0,C 180,E1 -18438.065,E2 -18438.065} C_VEL
LIN {X 0,Y 254.33,Z 621.643,A -85,B 0,C 180,E1 -18440.457,E2 -18440.457} C_VEL
LIN {X 0,Y 253.955,Z 624.169,A -85,B 0,C 180,E1 -18443.645,E2 -18443.645} C_VEL
LIN {X 0,Y 253.931,Z 625.516,A -85,B 0,C 180,E1 -18446.828,E2 -18446.828} C_VEL
LIN {X 0,Y 254.058,Z 625.656,A -85,B 0,C 180,E1 -18450.001,E2 -18450.001} C_VEL
LIN {X 0,Y 253.958,Z 624.621,A -85,B 0,C 180,E1 -18453.173,E2 -18453.173} C_VEL
LIN {X 0,Y 253.968,Z 622.39,A -85,B 0,C 180,E1 -18456.356,E2 -18456.356} C_VEL
LIN {X 0,Y 254.331,Z 618.917,A -85,B 0,C 180,E1 -18459.544,E2 -18459.544} C_VEL
LIN {X 0,Y 255.077,Z 614.104,A -85,B 0,C 180,E1 -18462.734,E2 -18462.734} C_VEL
LIN {X 0,Y 256.322,Z 607.82,A -85,B 0,C 180,E1 -18465.914,E2 -18465.914} C_VEL
LIN {X 0,Y 257.977,Z 600.992,A -85,B 0,C 180,E1 -18468.669,E2 -18468.669} C_VEL
LIN {X 0,Y 260.056,Z 592.722,A -85,B 0,C 180,E1 -18471.398,E2 -18471.398} C_VEL
LIN {X 0,Y 262.349,Z 584.302,A -85,B 0,C 180,E1 -18473.693,E2 -18473.693} C_VEL
LIN {X 0,Y 264.873,Z 574.403,A -85,B 0,C 180,E1 -18475.964,E2 -18475.964} C_VEL
LIN {X 0,Y 267.915,Z 562.64,A -85,B 0,C 180,E1 -18478.176,E2 -18478.176} C_VEL
LIN {X 0,Y 271.046,Z 549.649,A -85,B 0,C 180,E1 -18480.157,E2 -18480.157} C_VEL
LIN {X 0,Y 273.837,Z 536.79,A -85,B 0,C 180,E1 -18481.744,E2 -18481.744} C_VEL
LIN {X 0,Y 276.528,Z 522.344,A -85,B 0,C 180,E1 -18483.168,E2 -18483.168} C_VEL
LIN {X 0,Y 278.928,Z 507.1,A -85,B 0,C 180,E1 -18484.317,E2 -18484.317} C_VEL
LIN {X 0,Y 280.827,Z 492.026,A -85,B 0,C 180,E1 -18485.142,E2 -18485.142} C_VEL
LIN {X 0,Y 282.148,Z 476.478,A -85,B 0,C 180,E1 -18485.718,E2 -18485.718} C_VEL
LIN {X 0,Y 286.936,Z 374.586,A -85,B 0,C 180,E1 -18488.338,E2 -18488.338} C_VEL
LIN {X 0,Y 286.214,Z 370.7,A -85,B 0,C 180,E1 -18488.561,E2 -18488.561} C_VEL
LIN {X 0,Y 278.07,Z 351.868,A -85,B 0,C 180,E1 -18490.341,E2 -18490.341} C_VEL
LIN {X 0,Y 270.23,Z 335.531,A -85,B 0,C 180,E1 -18492.124,E2 -18492.124} C_VEL
LIN {X 0,Y 262.287,Z 320.812,A -85,B 0,C 180,E1 -18494.002,E2 -18494.002} C_VEL
LIN {X 0,Y 258.118,Z 313.207,A -85,B 0,C 180,E1 -18495.066,E2 -18495.066} C_VEL
LIN {X 0,Y 256.042,Z 306.216,A -85,B 0,C 180,E1 -18497.826,E2 -18497.826} C_VEL
LIN {X 0,Y 256.068,Z 306.204,A -85,B 0,C 180,E1 -18500.855,E2 -18500.855} C_VEL
LIN {X 0,Y 256.082,Z 306.197,A -85,B 0,C 180,E1 -18504.805,E2 -18504.805} C_VEL
LIN {X 0,Y 256.08,Z 306.211,A -85,B 0,C 180,E1 -18508.568,E2 -18508.568} C_VEL
LIN {X 0,Y 256.079,Z 306.209,A -85,B 0,C 180,E1 -18512.187,E2 -18512.187} C_VEL
LIN {X 0,Y 256.085,Z 306.211,A -85,B 0,C 180,E1 -18515.689,E2 -18515.689} C_VEL
LIN {X 0,Y 256.122,Z 306.212,A -85,B 0,C 180,E1 -18519.099,E2 -18519.099} C_VEL
LIN {X 0,Y 256.23,Z 306.19,A -85,B 0,C 180,E1 -18524.078,E2 -18524.078} C_VEL
LIN {X 0,Y 256.277,Z 306.156,A -85,B 0,C 180,E1 -18528.93,E2 -18528.93} C_VEL
LIN {X 0,Y 256.453,Z 306.165,A -85,B 0,C 180,E1 -18532.122,E2 -18532.122} C_VEL
LIN {X 0,Y 256.283,Z 306.156,A -85,B 0,C 180,E1 -18535.279,E2 -18535.279} C_VEL
LIN {X 0,Y 256.685,Z 306.107,A -85,B 0,C 180,E1 -18538.428,E2 -18538.428} C_VEL
LIN {X 0,Y 256.691,Z 306.137,A -85,B 0,C 180,E1 -18541.566,E2 -18541.566} C_VEL
LIN {X 0,Y 256.426,Z 306.122,A -85,B 0,C 180,E1 -18546.554,E2 -18546.554} C_VEL
LIN {X 0,Y 256.395,Z 306.157,A -85,B 0,C 180,E1 -18549.463,E2 -18549.463} C_VEL
LIN {X 0,Y 256.225,Z 306.176,A -85,B 0,C 180,E1 -18554.289,E2 -18554.289} C_VEL
LIN {X 0,Y 256.166,Z 306.157,A -85,B 0,C 180,E1 -18557.562,E2 -18557.562} C_VEL
LIN {X 0,Y 256.13,Z 306.201,A -85,B 0,C 180,E1 -18561.105,E2 -18561.105} C_VEL
LIN {X 0,Y 256.075,Z 306.187,A -85,B 0,C 180,E1 -18565.085,E2 -18565.085} C_VEL
LIN {X 0,Y 256.066,Z 306.18,A -85,B 0,C 180,E1 -18568.566,E2 -18568.566} C_VEL
LIN {X 0,Y 256.06,Z 306.215,A -85,B 0,C 180,E1 -18571.697,E2 -18571.697} C_VEL
LIN {X 0,Y 256.068,Z 306.186,A -85,B 0,C 180,E1 -18575.191,E2 -18575.191} C_VEL
LIN {X 0,Y 256.054,Z 306.201,A -85,B 0,C 180,E1 -18579.141,E2 -18579.141} C_VEL
LIN {X 0,Y 256.013,Z 306.208,A -85,B 0,C 180,E1 -18583.333,E2 -18583.333} C_VEL
LIN {X 0,Y 256.057,Z 306.208,A -85,B 0,C 180,E1 -18587.817,E2 -18587.817} C_VEL
LIN {X 0,Y 256.059,Z 306.208,A -85,B 0,C 180,E1 -18590.856,E2 -18590.856} C_VEL
LIN {X 0,Y 256.113,Z 306.184,A -85,B 0,C 180,E1 -18592.865,E2 -18592.865} C_VEL
LIN {X 0,Y 256.053,Z 306.219,A -85,B 0,C 180,E1 -18596.705,E2 -18596.705} C_VEL
LIN {X 0,Y 256.112,Z 306.201,A -85,B 0,C 180,E1 -18601.408,E2 -18601.408} C_VEL
LIN {X 0,Y 256.128,Z 306.193,A -85,B 0,C 180,E1 -18605.695,E2 -18605.695} C_VEL
LIN {X 0,Y 256.147,Z 306.193,A -85,B 0,C 180,E1 -18609.103,E2 -18609.103} C_VEL
LIN {X 0,Y 256.265,Z 306.181,A -85,B 0,C 180,E1 -18614.083,E2 -18614.083} C_VEL
LIN {X 0,Y 256.278,Z 306.186,A -85,B 0,C 180,E1 -18614.848,E2 -18614.848} C_VEL
LIN {X 0,Y 257.188,Z 308.908,A -85,B 0,C 180,E1 -18615.139,E2 -18615.139} C_VEL
LIN {X 0,Y 259.021,Z 311.335,A -85,B 0,C 180,E1 -18615.572,E2 -18615.572} C_VEL
LIN {X 0,Y 261.217,Z 314.739,A -85,B 0,C 180,E1 -18616.098,E2 -18616.098} C_VEL
LIN {X 0,Y 272.823,Z 333.429,A -85,B 0,C 180,E1 -18618.728,E2 -18618.728} C_VEL
LIN {X 0,Y 275.964,Z 339.374,A -85,B 0,C 180,E1 -18619.425,E2 -18619.425} C_VEL
LIN {X 0,Y 284.289,Z 356.704,A -85,B 0,C 180,E1 -18621.228,E2 -18621.228} C_VEL
LIN {X 0,Y 287.161,Z 363.53,A -85,B 0,C 180,E1 -18621.846,E2 -18621.846} C_VEL
LIN {X 0,Y 282.28,Z 465.638,A -85,B 0,C 180,E1 -18624.477,E2 -18624.477} C_VEL
LIN {X 0,Y 280.9,Z 481.689,A -85,B 0,C 180,E1 -18625.151,E2 -18625.151} C_VEL
LIN {X 0,Y 279.158,Z 496.134,A -85,B 0,C 180,E1 -18626.03,E2 -18626.03} C_VEL
LIN {X 0,Y 277.106,Z 509.436,A -85,B 0,C 180,E1 -18627.092,E2 -18627.092} C_VEL
LIN {X 0,Y 274.496,Z 524.212,A -85,B 0,C 180,E1 -18628.602,E2 -18628.602} C_VEL
LIN {X 0,Y 271.539,Z 538.005,A -85,B 0,C 180,E1 -18630.37,E2 -18630.37} C_VEL
LIN {X 0,Y 268.489,Z 550.92,A -85,B 0,C 180,E1 -18632.437,E2 -18632.437} C_VEL
LIN {X 0,Y 265.7,Z 561.745,A -85,B 0,C 180,E1 -18634.551,E2 -18634.551} C_VEL
LIN {X 0,Y 262.776,Z 572.744,A -85,B 0,C 180,E1 -18637.173,E2 -18637.173} C_VEL
LIN {X 0,Y 260.416,Z 581.433,A -85,B 0,C 180,E1 -18639.71,E2 -18639.71} C_VEL
LIN {X 0,Y 258.245,Z 589.47,A -85,B 0,C 180,E1 -18642.574,E2 -18642.574} C_VEL
LIN {X 0,Y 256.784,Z 595.182,A -85,B 0,C 180,E1 -18645.07,E2 -18645.07} C_VEL
LIN {X 0,Y 255.681,Z 600,A -85,B 0,C 180,E1 -18647.598,E2 -18647.598} C_VEL
LIN {X 0,Y 254.684,Z 604.995,A -85,B 0,C 180,E1 -18651.021,E2 -18651.021} C_VEL
LIN {X 0,Y 253.953,Z 608.551,A -85,B 0,C 180,E1 -18654.525,E2 -18654.525} C_VEL
LIN {X 0,Y 253.571,Z 610.669,A -85,B 0,C 180,E1 -18658.109,E2 -18658.109} C_VEL
LIN {X 0,Y 253.591,Z 611.279,A -85,B 0,C 180,E1 -18660.788,E2 -18660.788} C_VEL
LIN {X 0,Y 253.769,Z 611,A -85,B 0,C 180,E1 -18663.822,E2 -18663.822} C_VEL
LIN {X 0,Y 254.331,Z 609.315,A -85,B 0,C 180,E1 -18667.438,E2 -18667.438} C_VEL
LIN {X 0,Y 254.896,Z 607.704,A -85,B 0,C 180,E1 -18669.47,E2 -18669.47} C_VEL
LIN {X 0,Y 255.846,Z 604.863,A -85,B 0,C 180,E1 -18672.13,E2 -18672.13} C_VEL
LIN {X 0,Y 257.391,Z 600.394,A -85,B 0,C 180,E1 -18675.226,E2 -18675.226} C_VEL
LIN {X 0,Y 259.748,Z 593.779,A -85,B 0,C 180,E1 -18678.659,E2 -18678.659} C_VEL
LIN {X 0,Y 262.401,Z 586.597,A -85,B 0,C 180,E1 -18681.574,E2 -18681.574} C_VEL
LIN {X 0,Y 265.587,Z 577.897,A -85,B 0,C 180,E1 -18684.401,E2 -18684.401} C_VEL
LIN {X 0,Y 268.821,Z 568.883,A -85,B 0,C 180,E1 -18686.78,E2 -18686.78} C_VEL
LIN {X 0,Y 272.479,Z 558.045,A -85,B 0,C 180,E1 -18689.129,E2 -18689.129} C_VEL
LIN {X 0,Y 276.148,Z 546.328,A -85,B 0,C 180,E1 -18691.193,E2 -18691.193} C_VEL
LIN {X 0,Y 279.976,Z 532.665,A -85,B 0,C 180,E1 -18693.142,E2 -18693.142} C_VEL
LIN {X 0,Y 283.009,Z 520.406,A -85,B 0,C 180,E1 -18694.543,E2 -18694.543} C_VEL
LIN {X 0,Y 285.961,Z 506.319,A -85,B 0,C 180,E1 -18695.837,E2 -18695.837} C_VEL
LIN {X 0,Y 288.461,Z 491.534,A -85,B 0,C 180,E1 -18696.882,E2 -18696.882} C_VEL
LIN {X 0,Y 290.491,Z 476.105,A -85,B 0,C 180,E1 -18697.667,E2 -18697.667} C_VEL
LIN {X 0,Y 291.823,Z 460.21,A -85,B 0,C 180,E1 -18698.207,E2 -18698.207} C_VEL
LIN {X 0,Y 297.002,Z 369.849,A -85,B 0,C 180,E1 -18700.523,E2 -18700.523} C_VEL
LIN {X 0,Y 294.513,Z 364.363,A -85,B 0,C 180,E1 -18701.246,E2 -18701.246} C_VEL
LIN {X 0,Y 291.998,Z 360.384,A -85,B 0,C 180,E1 -18701.941,E2 -18701.941} C_VEL
LIN {X 0,Y 288.944,Z 357.31,A -85,B 0,C 180,E1 -18702.748,E2 -18702.748} C_VEL
LIN {X 0,Y 281.634,Z 350.927,A -85,B 0,C 180,E1 -18704.784,E2 -18704.784} C_VEL
LIN {X 0,Y 279.129,Z 347.273,A -85,B 0,C 180,E1 -18705.603,E2 -18705.603} C_VEL
LIN {X 0,Y 275.246,Z 340.993,A -85,B 0,C 180,E1 -18706.995,E2 -18706.995} C_VEL
LIN {X 0,Y 271.449,Z 335.644,A -85,B 0,C 180,E1 -18708.42,E2 -18708.42} C_VEL
LIN {X 0,Y 269.124,Z 332.438,A -85,B 0,C 180,E1 -18709.339,E2 -18709.339} C_VEL
LIN {X 0,Y 265.709,Z 327.923,A -85,B 0,C 180,E1 -18710.78,E2 -18710.78} C_VEL
LIN {X 0,Y 263.13,Z 324.388,A -85,B 0,C 180,E1 -18711.977,E2 -18711.977} C_VEL
LIN {X 0,Y 262.364,Z 323.299,A -85,B 0,C 180,E1 -18712.348,E2 -18712.348} C_VEL
LIN {X 0,Y 259.833,Z 320.491,A -85,B 0,C 180,E1 -18713.572,E2 -18713.572} C_VEL
LIN {X 0,Y 258.591,Z 318.403,A -85,B 0,C 180,E1 -18714.251,E2 -18714.251} C_VEL
LIN {X 0,Y 255.916,Z 316.253,A -85,B 0,C 180,E1 -18715.672,E2 -18715.672} C_VEL
LIN {X 0,Y 254.371,Z 313.463,A -85,B 0,C 180,E1 -18716.686,E2 -18716.686} C_VEL
LIN {X 0,Y 254.178,Z 312.917,A -85,B 0,C 180,E1 -18716.833,E2 -18716.833} C_VEL
LIN {X 0,Y 251.64,Z 311.101,A -85,B 0,C 180,E1 -18718.402,E2 -18718.402} C_VEL
LIN {X 0,Y 250.172,Z 308.831,A -85,B 0,C 180,E1 -18719.5,E2 -18719.5} C_VEL
LIN {X 0,Y 249.719,Z 307.001,A -85,B 0,C 180,E1 -18720.003,E2 -18720.003} C_VEL
LIN {X 0,Y 249.419,Z 307.041,A -85,B 0,C 180,E1 -18723.233,E2 -18723.233} C_VEL
LIN {X 0,Y 249.428,Z 307.042,A -85,B 0,C 180,E1 -18726.474,E2 -18726.474} C_VEL
LIN {X 0,Y 249.327,Z 307.053,A -85,B 0,C 180,E1 -18729.74,E2 -18729.74} C_VEL
LIN {X 0,Y 249.165,Z 307.067,A -85,B 0,C 180,E1 -18734.708,E2 -18734.708} C_VEL
LIN {X 0,Y 249.09,Z 307.079,A -85,B 0,C 180,E1 -18738.083,E2 -18738.083} C_VEL
LIN {X 0,Y 249.039,Z 307.09,A -85,B 0,C 180,E1 -18741.525,E2 -18741.525} C_VEL
LIN {X 0,Y 249.041,Z 307.082,A -85,B 0,C 180,E1 -18745.443,E2 -18745.443} C_VEL
LIN {X 0,Y 249.054,Z 307.272,A -85,B 0,C 180,E1 -18747.524,E2 -18747.524} C_VEL
LIN {X 0,Y 249.957,Z 309.846,A -85,B 0,C 180,E1 -18750.083,E2 -18750.083} C_VEL
LIN {X 0,Y 254.96,Z 316.153,A -85,B 0,C 180,E1 -18753.459,E2 -18753.459} C_VEL
LIN {X 0,Y 256.104,Z 317.747,A -85,B 0,C 180,E1 -18754.161,E2 -18754.161} C_VEL
LIN {X 0,Y 260.875,Z 324.114,A -85,B 0,C 180,E1 -18756.724,E2 -18756.724} C_VEL
LIN {X 0,Y 265.02,Z 330.232,A -85,B 0,C 180,E1 -18758.727,E2 -18758.727} C_VEL
LIN {X 0,Y 269.31,Z 336.634,A -85,B 0,C 180,E1 -18760.57,E2 -18760.57} C_VEL
LIN {X 0,Y 274.873,Z 345.596,A -85,B 0,C 180,E1 -18762.749,E2 -18762.749} C_VEL
LIN {X 0,Y 281.635,Z 357.881,A -85,B 0,C 180,E1 -18765.152,E2 -18765.152} C_VEL
LIN {X 0,Y 287.271,Z 369.724,A -85,B 0,C 180,E1 -18767.015,E2 -18767.015} C_VEL
LIN {X 0,Y 291.67,Z 380.295,A -85,B 0,C 180,E1 -18768.399,E2 -18768.399} C_VEL
LIN {X 0,Y 285.6,Z 479.769,A -85,B 0,C 180,E1 -18771.023,E2 -18771.023} C_VEL
LIN {X 0,Y 283.69,Z 495.639,A -85,B 0,C 180,E1 -18771.677,E2 -18771.677} C_VEL
LIN {X 0,Y 281.065,Z 510.837,A -85,B 0,C 180,E1 -18772.562,E2 -18772.562} C_VEL
LIN {X 0,Y 278.325,Z 524.142,A -85,B 0,C 180,E1 -18773.603,E2 -18773.603} C_VEL
LIN {X 0,Y 274.97,Z 537.717,A -85,B 0,C 180,E1 -18774.955,E2 -18774.955} C_VEL
LIN {X 0,Y 271.33,Z 550.82,A -85,B 0,C 180,E1 -18776.606,E2 -18776.606} C_VEL
LIN {X 0,Y 267.448,Z 563.131,A -85,B 0,C 180,E1 -18778.517,E2 -18778.517} C_VEL
LIN {X 0,Y 263.231,Z 575.287,A -85,B 0,C 180,E1 -18780.841,E2 -18780.841} C_VEL
LIN {X 0,Y 259.504,Z 585.804,A -85,B 0,C 180,E1 -18783.348,E2 -18783.348} C_VEL
LIN {X 0,Y 256.09,Z 595.241,A -85,B 0,C 180,E1 -18786.123,E2 -18786.123} C_VEL
LIN {X 0,Y 253.215,Z 602.802,A -85,B 0,C 180,E1 -18788.851,E2 -18788.851} C_VEL
LIN {X 0,Y 250.628,Z 609.903,A -85,B 0,C 180,E1 -18792.035,E2 -18792.035} C_VEL
LIN {X 0,Y 248.866,Z 615.537,A -85,B 0,C 180,E1 -18795.277,E2 -18795.277} C_VEL
LIN {X 0,Y 247.626,Z 619.848,A -85,B 0,C 180,E1 -18798.542,E2 -18798.542} C_VEL
LIN {X 0,Y 247.019,Z 622.924,A -85,B 0,C 180,E1 -18801.822,E2 -18801.822} C_VEL
LIN {X 0,Y 246.809,Z 624.893,A -85,B 0,C 180,E1 -18805.323,E2 -18805.323} C_VEL
LIN {X 0,Y 246.922,Z 625.538,A -85,B 0,C 180,E1 -18808.37,E2 -18808.37} C_VEL
LIN {X 0,Y 246.987,Z 625.442,A -85,B 0,C 180,E1 -18810.001,E2 -18810.001} C_VEL
LIN {X 0,Y 246.858,Z 624.364,A -85,B 0,C 180,E1 -18813.265,E2 -18813.265} C_VEL
LIN {X 0,Y 246.884,Z 622.09,A -85,B 0,C 180,E1 -18816.539,E2 -18816.539} C_VEL
LIN {X 0,Y 247.287,Z 618.569,A -85,B 0,C 180,E1 -18819.819,E2 -18819.819} C_VEL
LIN {X 0,Y 248.077,Z 613.703,A -85,B 0,C 180,E1 -18823.1,E2 -18823.1} C_VEL
LIN {X 0,Y 249.385,Z 607.358,A -85,B 0,C 180,E1 -18826.369,E2 -18826.369} C_VEL
LIN {X 0,Y 251.153,Z 600.492,A -85,B 0,C 180,E1 -18829.196,E2 -18829.196} C_VEL
LIN {X 0,Y 253.374,Z 592.155,A -85,B 0,C 180,E1 -18831.991,E2 -18831.991} C_VEL
LIN {X 0,Y 255.756,Z 583.65,A -85,B 0,C 180,E1 -18834.343,E2 -18834.343} C_VEL
LIN {X 0,Y 258.418,Z 573.652,A -85,B 0,C 180,E1 -18836.663,E2 -18836.663} C_VEL
LIN {X 0,Y 261.624,Z 561.776,A -85,B 0,C 180,E1 -18838.916,E2 -18838.916} C_VEL
LIN {X 0,Y 264.549,Z 549.951,A -85,B 0,C 180,E1 -18840.757,E2 -18840.757} C_VEL
LIN {X 0,Y 267.424,Z 537.203,A -85,B 0,C 180,E1 -18842.375,E2 -18842.375} C_VEL
LIN {X 0,Y 270.098,Z 523.543,A -85,B 0,C 180,E1 -18843.769,E2 -18843.769} C_VEL
LIN {X 0,Y 272.496,Z 509.195,A -85,B 0,C 180,E1 -18844.907,E2 -18844.907} C_VEL
LIN {X 0,Y 274.541,Z 494.127,A -85,B 0,C 180,E1 -18845.787,E2 -18845.787} C_VEL
LIN {X 0,Y 275.88,Z 479.947,A -85,B 0,C 180,E1 -18846.376,E2 -18846.376} C_VEL
LIN {X 0,Y 281.026,Z 375.647,A -85,B 0,C 180,E1 -18849.118,E2 -18849.118} C_VEL
LIN {X 0,Y 280.533,Z 373.44,A -85,B 0,C 180,E1 -18849.261,E2 -18849.261} C_VEL
LIN {X 0,Y 272.053,Z 353.636,A -85,B 0,C 180,E1 -18851.2,E2 -18851.2} C_VEL
LIN {X 0,Y 264.635,Z 338.387,A -85,B 0,C 180,E1 -18852.944,E2 -18852.944} C_VEL
LIN {X 0,Y 256.004,Z 322.209,A -85,B 0,C 180,E1 -18855.085,E2 -18855.085} C_VEL
LIN {X 0,Y 250.759,Z 313.003,A -85,B 0,C 180,E1 -18856.47,E2 -18856.47} C_VEL
LIN {X 0,Y 248.993,Z 307.098,A -85,B 0,C 180,E1 -18858.983,E2 -18858.983} C_VEL
LIN {X 0,Y 249.047,Z 307.089,A -85,B 0,C 180,E1 -18862.199,E2 -18862.199} C_VEL
LIN {X 0,Y 249.046,Z 307.07,A -85,B 0,C 180,E1 -18865.637,E2 -18865.637} C_VEL
LIN {X 0,Y 248.996,Z 307.09,A -85,B 0,C 180,E1 -18869.463,E2 -18869.463} C_VEL
LIN {X 0,Y 249.015,Z 307.087,A -85,B 0,C 180,E1 -18873.153,E2 -18873.153} C_VEL
LIN {X 0,Y 249.006,Z 307.09,A -85,B 0,C 180,E1 -18876.723,E2 -18876.723} C_VEL
LIN {X 0,Y 249.047,Z 307.085,A -85,B 0,C 180,E1 -18880.204,E2 -18880.204} C_VEL
LIN {X 0,Y 249.158,Z 307.074,A -85,B 0,C 180,E1 -18883.614,E2 -18883.614} C_VEL
LIN {X 0,Y 249.183,Z 307.028,A -85,B 0,C 180,E1 -18886.957,E2 -18886.957} C_VEL
LIN {X 0,Y 249.372,Z 307.039,A -85,B 0,C 180,E1 -18890.536,E2 -18890.536} C_VEL
LIN {X 0,Y 249.417,Z 307.035,A -85,B 0,C 180,E1 -18893.526,E2 -18893.526} C_VEL
LIN {X 0,Y 249.644,Z 306.982,A -85,B 0,C 180,E1 -18898.384,E2 -18898.384} C_VEL
LIN {X 0,Y 249.652,Z 307.014,A -85,B 0,C 180,E1 -18901.61,E2 -18901.61} C_VEL
LIN {X 0,Y 249.405,Z 306.996,A -85,B 0,C 180,E1 -18906.53,E2 -18906.53} C_VEL
LIN {X 0,Y 249.328,Z 307.04,A -85,B 0,C 180,E1 -18909.734,E2 -18909.734} C_VEL
LIN {X 0,Y 249.168,Z 307.047,A -85,B 0,C 180,E1 -18914.703,E2 -18914.703} C_VEL
LIN {X 0,Y 249.101,Z 307.04,A -85,B 0,C 180,E1 -18918.077,E2 -18918.077} C_VEL
LIN {X 0,Y 249.07,Z 307.085,A -85,B 0,C 180,E1 -18921.516,E2 -18921.516} C_VEL
LIN {X 0,Y 249.036,Z 307.058,A -85,B 0,C 180,E1 -18925.437,E2 -18925.437} C_VEL
LIN {X 0,Y 249.014,Z 307.064,A -85,B 0,C 180,E1 -18928.965,E2 -18928.965} C_VEL
